Omron CX-Programmer project NewProject (CX-Programmer 9.51)

# PLC NewPLC1: CJ2M CPU11
I/O table (CPU CJ2M-CPU11): rack 0 slot 0 CJ1W-ID211; rack 0 slot 1 CJ1W-OD212; rack 0 slot 2 CJ1W-TC002; rack 0 slot 3 CJ1W-TC002; rack 0 slot 4 CJ1W-NC481; rack 0 slot 5 CJ1W-DA041; rack 0 slot 6 CJ1W-MAD42

## Global symbols (name address type ; comment)
AUX_AUTOMATICO W10.00 BOOL  ; Auxiliar maquina em Automático
AUX_LIMITE_NIPE W4.00 BOOL
AUX_MANUAL W10.01 BOOL  ; auxiliar maquina em trabalho manual
AUX_MANUAL_SERVO_NIP_LOCK W20.00 BOOL  ; Auxiliar para ligar manual do servo NIP
AUX_MANUAL_SERVO_NIP_UNLOCK W20.09 BOOL  ; Auxiliar UNLOCK servo NIP
AUX_MANUAL_SERVO_SEL_LOCK W20.02 BOOL  ; Auxiliar par ligar servo SEL
AUX_MANUAL_SERVO_SEL_UNLOCK W20.11 BOOL  ; Auxiliar para UNLOCK Servo SEL
AUX_MANUAL_SERVO_TRO_LOCK W20.01 BOOL  ; Auxiliar  para ligar servo TRO
AUX_MANUAL_SERVO_TRO_UNLOCK W20.10 BOOL  ; Auxiliar Unlock servo TRO
0.05 BOOL  ; Chave seletora Faca
0.13 BOOL  ; Botão Jog FACA avança
1.05 BOOL  ; INVERSOR DE PASSAGEM
1.12 BOOL  ; Saida habilita servo rebobinador inferior 2
1.13 BOOL  ; Saida Habililta servo rebobinador superior 2
2000.00 BOOL  ; Habilita Saída analógica 1
2000.01 BOOL  ; Habilita saída analógica 2
2030.00 BOOL  ; Habilita saída Rebobinador Superior 1
2030.01 BOOL  ; Habilita saída Rebobinador inferior 1
2030.02 BOOL  ; Habilita saída Rebobinador Superior 2
2030.03 BOOL  ; Habilita saída Rebobinador Inferior 2
2031 CHANNEL  ; Saída Analógica Rebobinador Superior
2032 CHANNEL  ; Saída Analógica Rebobinador  Inferior 1
2033 CHANNEL  ; Habilita saída Rebobinador Superior 2
2034 CHANNEL  ; Saída Analógica Rebobinador  Inferior 2
2040 CHANNEL  ; Setpoint da saída de aquecimento 5
A531.00 BOOL  ; ZERA CONTAGEM DO SENSOR
A531.01 BOOL  ; ZERA
D1012 CHANNEL  ; Posição do Corte
D1014 CHANNEL  ; Posição corte inferior
D104 CHANNEL  ; Valor para saida analógica reb sup 2
D106 CHANNEL  ; valor desejado de saida para rebobinador inferior 2
D124 CHANNEL  ; PRESET VALOR MIN DO TORQUE REB SUP 2
D126 CHANNEL  ; IHM preset valor min de torque para trabalho inferior2
D20 CHANNEL  ; CONT ETIQUETA
D200 CHANNEL  ; Controle Desbobinador Superior
D201 CHANNEL  ; Banda Proporcional Desbobinador superior
D202 CHANNEL  ; Constante Integral Desbobinador Superior
D203 CHANNEL  ; Constante Derivativo Desbobinador Superior
D204 CHANNEL  ; Tempo de Amostragem
D205 CHANNEL  ; Controle PID Desbobinador Sup
D206 CHANNEL  ; Controle PID Desbobinador Sup
D207 CHANNEL  ; Limite da variável manipulada
D209 CHANNEL  ; Controle PID automático e ganho
D210 CHANNEL  ; Histerese
D280 CHANNEL  ; Set Point Desbobinador Superior
D403 CHANNEL  ; IHM Constante selagem
D404 CHANNEL  ; IHM Constante Faca
D405 CHANNEL  ; FREIO DESBOBINADOR SUPERIOR
D406 CHANNEL  ; IHM Freio Desbobinador Inferior
D408 CHANNEL  ; IHM Tamanho do Pacote
D410 CHANNEL  ; IHM Velocidade Maquina M/min
D54 CHANNEL  ; IHM preset torque do Reb Sup 2, quando em automatico
D56 CHANNEL  ; IHM preset para torque Reb inf 2 quando a maquina estiver em trabalho
D700 CHANNEL  ; CONTANTE ACELERACAO
D701 CHANNEL  ; VELOCIDADE_ETQ
H0.00 BOOL  ; Seletora quantidade de facas
H45.00 BOOL  ; HABILITA ETIQUETA
T0002 BOOL  ; Tempo para acionamento do marcador
T0021 BOOL  ; Tempo para Reset
T0050 BOOL  ; ]
T0100 BOOL  ; Tempo Reset Ethercat
T0101 BOOL  ; Tempo para iniciar a verificação se chegou na origem
W1.00 BOOL  ; INDICA SERVOS LIGADOS
W1.02 BOOL  ; FLAG EM PRODUÇÃO
W1.03 BOOL  ; TRO REFERENCIADO
W200.00 BOOL  ; Aumento gradativo do torque
W20.03 BOOL  ; Auxiliar JOG NIP Horario
W20.04 BOOL  ; Auxiliar JOG NIP Anti-horario
W20.05 BOOL  ; Auxiliar JOG TRO Horario
W20.06 BOOL  ; Auxiliar JOG TRO Anti Horario
W20.07 BOOL  ; Auxiliar JOG SEL Horario
W20.08 BOOL  ; Auxiliar JOG SEL Anti horario
W2.03 BOOL  ; Auxiliar servos não estão em erro
W2.04 BOOL  ; Auxiliar Servos Lock
W2.05 BOOL  ; Auxiliar busca de origem
W33.00 BOOL  ; +
W33.01 BOOL  ; -
W3.00 BOOL  ; Flag Inicialização Completa
W50.07 BOOL  ; IHM botão liga servo Selagem
W50.08 BOOL  ; IHM botão liga servo TRO
W50.09 BOOL  ; IHM Botão Liga servo NIP Manual
W50.10 BOOL  ; IHM botão JOG SEL Horario
W50.11 BOOL  ; IHM botão JOG SEL Anti Horario
W50.12 BOOL  ; IHM botão JOG TRO Horario
W50.13 BOOL  ; IHM botão JOG TRO Anti Horario
W50.14 BOOL  ; IHM botão JOG NIP Horario
W50.15 BOOL  ; IHM botão JOG NIP Anti Horario
W60.04 BOOL  ; Botão Habilita servo Rebobinador superior 2
W60.05 BOOL  ; Botão Habilita servo Rebobinador inferior 2
W60.09 BOOL  ; IHM  Botão Reset
W60.10 BOOL  ; IHM PB busca da origem servo TRO
W60.11 BOOL  ; IHM Botão Liga/Desliga todos servos
W6.00 BOOL  ; PARA ROLDANA
W6.08 BOOL  ; SALVAR RECEITA
W6.09 BOOL  ; CARREGAR RECEITA
W6.12 BOOL  ; FLAG PERCA CORTE
W6.14 BOOL  ; MARCAR SENSOR
W7.00 BOOL  ; START AT1
W7.01 BOOL  ; START AT2
W7.02 BOOL  ; START AT3
W7.03 BOOL  ; START AT4
W7.04 BOOL  ; START AT5
W8.00 BOOL  ; MARCA SENSOR ETIQUETA
CH_SEL_LIGA_NIP 0.04 BOOL  ; Chave seletora para ligar acionamento do NIP
CH_SEL_MANUAL_AUTO 0.03 BOOL  ; Chave de seleção Manual ou Automático
CONTAGEM_ABS D670 CHANNEL  ; CONTAGEM_ABS
Calc_Sel Calc_Pacote
Calc_Tamanho_Pacote Calc_Pacote
Desbobinador_Sup Escala_SA
ETIQUETADOR CALC_ETIQUETA
IHM_Auto_Torque_Reb_Inf D52 REAL  ; IHM preset para torque rebobinador inferior quando a maquina estiver em trabalho
IHM_Auto_Torque_Reb_Sup D50 REAL  ; IHM preset torque do Rebobinador Superior, quando em automático
IHM_BT_FREIO_INF W60.01 BOOL
IHM_BT_FREIO_SUP W60.00 BOOL  ; Botão para acionamento no freio manual
IHM_BT_LOCK_REB_INF W60.03 BOOL  ; Botão Habilita servo Rebobinador inferior 1
IHM_BT_LOCK_REB_SUP W60.02 BOOL  ; Botão Habilita servo Rebobinador superior 1
IHM_Min_Reb_Inf D122 REAL  ; IHM preset valor minimo de torque para trabalho
IHM_Min_Reb_Sup D120 REAL  ; PRESET VALOR MINIMO DO TORQUE
IHM_PB_S_MARCADOR W50.03 BOOL  ; IHM Botão Acionamento manual do Etiquetador
IHM_PB_S_NIP W50.00 BOOL  ; IHM Botão acionamento manual do NIP
IHM_PB_S_NIP_SEL W50.02 BOOL  ; NIP Selagem
IHM_PB_S_SEL W50.01 BOOL  ; IHM Botão acionamento manual do tracionador Selagem
Inicializacao W0 CHANNEL  ; Controle inicialização
Inicializacao_passo_0 W0.00 BOOL
Inicializacao_passo_1 W0.01 BOOL
Inicializacao_passo_10 W0.10 BOOL
Inicializacao_passo_11 W0.11 BOOL
Inicializacao_passo_12 W0.12 BOOL
Inicializacao_passo_13 W0.13 BOOL
Inicializacao_passo_14 W0.14 BOOL
Inicializacao_passo_15 W0.15 BOOL
Inicializacao_passo_2 W0.02 BOOL
Inicializacao_passo_3 W0.03 BOOL
Inicializacao_passo_4 W0.04 BOOL
Inicializacao_passo_5 W0.05 BOOL
Inicializacao_passo_6 W0.06 BOOL
Inicializacao_passo_7 W0.07 BOOL
Inicializacao_passo_8 W0.08 BOOL
Inicializacao_passo_9 W0.09 BOOL
NCx8x_00_Axis1DirectOperation_AbsoluteMovementBit 3100.00 BOOL  ; AbsoluteMovementBit
NCx8x_00_Axis1DirectOperation_AccelerationTime 3108 DINT  ; AccelerationTime
NCx8x_00_Axis1DirectOperation_CommandPosition 3102 DINT  ; CommandPosition
NCx8x_00_Axis1DirectOperation_CommandSpeed 3104 DINT  ; CommandSpeed
NCx8x_00_Axis1DirectOperation_DecelerationTime 3110 DINT  ; DecelerationTime
NCx8x_00_Axis1DirectOperation_InterruptFeedingSpecificationBit 3100.05 BOOL  ; InterruptFeedingSpecificationBit
NCx8x_00_Axis1DirectOperation_InterruptInputMask_PresentPositionLatchEnableBit 3100.06 BOOL  ; InterruptInputMask_PresentPositionLatchEnableBit
NCx8x_00_Axis1DirectOperation_LatchCompletedFlagClearBit 3100.15 BOOL  ; LatchCompletedFlagClearBit
NCx8x_00_Axis1DirectOperation_OptionInput1 3106 UINT  ; OptionInput1
NCx8x_00_Axis1DirectOperation_OptionInput2 3107 UINT  ; OptionInput2
NCx8x_00_Axis1DirectOperation_OriginPositionLachCompletedFlagClearBit 3100.14 BOOL  ; OriginPositionLachCompletedFlagClearBit
NCx8x_00_Axis1DirectOperation_OriginPositionLachEnableBit 3100.11 BOOL  ; OriginPositionLachEnableBit
NCx8x_00_Axis1DirectOperation_PresentPositionPresetBit 3100.07 BOOL  ; PresentPositionPresetBit
NCx8x_00_Axis1DirectOperation_RelativeMovementBit 3100.01 BOOL  ; RelativeMovementBit
NCx8x_00_Axis1DirectOperation_RotationAxisDirection 3101 UINT  ; RotationAxisDirection
NCx8x_00_Axis1DirectOperation_SpeedControlBit 3100.02 BOOL  ; SpeedControlBit
NCx8x_00_Axis1ExpandedMonitor_ExpandedMonitor2 3500 DINT  ; ExpandedMonitor2
NCx8x_00_Axis1ExpandedMonitor_ExpandedMonitor3 3502 DINT  ; ExpandedMonitor3
NCx8x_00_Axis1ExpandedMonitor_ExpandedMonitor4 3504 DINT  ; ExpandedMonitor4
NCx8x_00_Axis1ExpandedMonitor_ExpandedMonitor5 3506 DINT  ; ExpandedMonitor5
NCx8x_00_Axis1ExpandedMonitor_ExpandedMonitor6 3508 DINT  ; ExpandedMonitor6
NCx8x_00_Axis1ManualOperation_DecelerationStopBit 3000.14 BOOL  ; DecelerationStopBit
NCx8x_00_Axis1ManualOperation_DeviationCounterResetBit 3000.02 BOOL  ; DeviationCounterResetBit
NCx8x_00_Axis1ManualOperation_DriveAlarmResetBit 3000.01 BOOL  ; DriveAlarmResetBit
NCx8x_00_Axis1ManualOperation_ForwardJogging_InchingBit 3000.07 BOOL  ; ForwardJogging_InchingBit
NCx8x_00_Axis1ManualOperation_ForwardTorqueLimitBit 3000.03 BOOL  ; ForwardTorqueLimitBit
NCx8x_00_Axis1ManualOperation_ImmediateStopBit 3000.13 BOOL  ; ImmediateStopBit
NCx8x_00_Axis1ManualOperation_Jogging_InchingSpeedSelectionBit 3000.06 BOOL  ; Jogging_InchingSpeedSelectionBit
NCx8x_00_Axis1ManualOperation_OriginReturnBit 3000.11 BOOL  ; OriginReturnBit
NCx8x_00_Axis1ManualOperation_OriginSearchBit 3000.10 BOOL  ; OriginSearchBit
NCx8x_00_Axis1ManualOperation_Override 3001 UINT  ; Override
NCx8x_00_Axis1ManualOperation_OverrideEnableBit 3000.05 BOOL  ; OverrideEnableBit
NCx8x_00_Axis1ManualOperation_ReverseJogging_InchingBit 3000.08 BOOL  ; ReverseJogging_InchingBit
NCx8x_00_Axis1ManualOperation_ReverseTorqueLimitBit 3000.04 BOOL  ; ReverseTorqueLimitBit
NCx8x_00_Axis1ManualOperation_ServoLockBit 3000.00 BOOL  ; ServoLockBit
NCx8x_00_Axis1ManualOperation_ServoUnlockBit 3000.15 BOOL  ; ServoUnlockBit
NCx8x_00_Axis1Status_AbsoluteMovementAcknowledgedFlag 3301.00 BOOL  ; AbsoluteMovementAcknowledgedFlag
NCx8x_00_Axis1Status_AbsoluteMovementFlag 3304.04 BOOL  ; AbsoluteMovementFlag
NCx8x_00_Axis1Status_AccelerationFlag 3303.03 BOOL  ; AccelerationFlag
NCx8x_00_Axis1Status_AlarmResetOutputFlag 3306.01 BOOL  ; AlarmResetOutputFlag
NCx8x_00_Axis1Status_AxisBusyFlag 3302.00 BOOL  ; AxisBusyFlag
NCx8x_00_Axis1Status_AxisErrorFlag 3305.12 BOOL  ; AxisErrorFlag
NCx8x_00_Axis1Status_AxisWarningFlag 3305.11 BOOL  ; AxisWarningFlag
NCx8x_00_Axis1Status_CommandPresentPosition 3308 DINT  ; CommandPresentPosition
NCx8x_00_Axis1Status_CommandPresentPositionOverflowFlag 3305.04 BOOL  ; CommandPresentPositionOverflowFlag
NCx8x_00_Axis1Status_CommandPresentPositionUnderflowFlag 3305.05 BOOL  ; CommandPresentPositionUnderflowFlag
NCx8x_00_Axis1Status_ConstantSpeedFlag 3303.04 BOOL  ; ConstantSpeedFlag
NCx8x_00_Axis1Status_DecelerationFlag 3303.05 BOOL  ; DecelerationFlag
NCx8x_00_Axis1Status_DecelerationStopAcknowledgedFlag 3300.14 BOOL  ; DecelerationStopAcknowledgedFlag
NCx8x_00_Axis1Status_DecelerationStopFlag 3303.08 BOOL  ; DecelerationStopFlag
NCx8x_00_Axis1Status_DeviationCounterResetAcknowledgedFlag 3300.02 BOOL  ; DeviationCounterResetAcknowledgedFlag
NCx8x_00_Axis1Status_DeviationCounterResetInvalidFlag 3302.09 BOOL  ; DeviationCounterResetInvalidFlag
NCx8x_00_Axis1Status_DeviationCounterResetOutputFlag 3306.02 BOOL  ; DeviationCounterResetOutputFlag
NCx8x_00_Axis1Status_DirectOperationEnabledFlag 3302.02 BOOL  ; DirectOperationEnabledFlag
NCx8x_00_Axis1Status_DriveAlarmInputFlag 3306.15 BOOL  ; DriveAlarmInputFlag
NCx8x_00_Axis1Status_DriveAlarmResetAcknowledgedFlag 3300.01 BOOL  ; DriveAlarmResetAcknowledgedFlag
NCx8x_00_Axis1Status_EmergencyStopInputFlag 3306.13 BOOL  ; EmergencyStopInputFlag
NCx8x_00_Axis1Status_ErrorCode 3307 UINT  ; ErrorCode
NCx8x_00_Axis1Status_ExecutionErrorFlag 3305.10 BOOL  ; ExecutionErrorFlag
NCx8x_00_Axis1Status_ExpandedMonitor 3310 DINT  ; ExpandedMonitor
NCx8x_00_Axis1Status_FeedbackPresentPositionOverflowFlag 3305.06 BOOL  ; FeedbackPresentPositionOverflowFlag
NCx8x_00_Axis1Status_FeedbackPresentPositionUnderflowFlag 3305.07 BOOL  ; FeedbackPresentPositionUnderflowFlag
NCx8x_00_Axis1Status_ForwardJogging_InchingAcknowledgedFlag 3300.07 BOOL  ; ForwardJogging_InchingAcknowledgedFlag
NCx8x_00_Axis1Status_ForwardLimitInputFlag 3306.08 BOOL  ; ForwardLimitInputFlag
NCx8x_00_Axis1Status_ForwardTorqueLimitAcknowledgedFlag 3300.03 BOOL  ; ForwardTorqueLimitAcknowledgedFlag
NCx8x_00_Axis1Status_ForwardTorqueLimitOutputFlag 3306.03 BOOL  ; ForwardTorqueLimitOutputFlag
NCx8x_00_Axis1Status_HighSpeedPTPStartAcknowledgedFlag 3302.07 BOOL  ; HighSpeedPTPStartAcknowledgedFlag
NCx8x_00_Axis1Status_ImmediateStopAcknowledgedFlag 3300.13 BOOL  ; ImmediateStopAcknowledgedFlag
NCx8x_00_Axis1Status_ImmediateStopFlag 3303.09 BOOL  ; ImmediateStopFlag
NCx8x_00_Axis1Status_InterruptFeedingSpecificationAcknowledgedFlag 3301.05 BOOL  ; InterruptFeedingSpecificationAcknowledgedFlag
NCx8x_00_Axis1Status_InterruptFeeding_InterruptInputWaitingFlag 3304.07 BOOL  ; InterruptFeeding_InterruptInputWaitingFlag
NCx8x_00_Axis1Status_InterruptFeeding_PositioningFlag 3304.08 BOOL  ; InterruptFeeding_PositioningFlag
NCx8x_00_Axis1Status_InterruptInputFlag 3306.12 BOOL  ; InterruptInputFlag
NCx8x_00_Axis1Status_InterruptInputMask_PresentPositionLatchEnableAcknowledgedFlag 3301.06 BOOL  ; InterruptInputMask_PresentPositionLatchEnableAcknowledgedFlag
NCx8x_00_Axis1Status_JoggingEnabledFlag 3302.01 BOOL  ; JoggingEnabledFlag
NCx8x_00_Axis1Status_Jogging_InchingFlag 3304.03 BOOL  ; Jogging_InchingFlag
NCx8x_00_Axis1Status_Jogging_InchingSpeedSelectionAcknowledgedFlag 3300.06 BOOL  ; Jogging_InchingSpeedSelectionAcknowledgedFlag
NCx8x_00_Axis1Status_LatchCompletedFlag 3305.02 BOOL  ; LatchCompletedFlag
NCx8x_00_Axis1Status_LatchCompletedFlagClearAcknowledgedFlag 3301.15 BOOL  ; LatchCompletedFlagClearAcknowledgedFlag
NCx8x_00_Axis1Status_MainCircuitStatusFlag 3306.05 BOOL  ; MainCircuitStatusFlag
NCx8x_00_Axis1Status_MemoryOperationFlag 3304.11 BOOL  ; MemoryOperationFlag
NCx8x_00_Axis1Status_OriginDefinedFlag 3305.00 BOOL  ; OriginDefinedFlag
NCx8x_00_Axis1Status_OriginInputFlag 3306.11 BOOL  ; OriginInputFlag
NCx8x_00_Axis1Status_OriginPositionLatchCompletedFlag 3305.03 BOOL  ; OriginPositionLatchCompletedFlag
NCx8x_00_Axis1Status_OriginPositionLatchCompletedFlagClearAcknowledgedFlag 3301.14 BOOL  ; OriginPositionLatchCompletedFlagClearAcknowledgedFlag
NCx8x_00_Axis1Status_OriginPositionLatchEnableAcknowledgedFlag 3301.11 BOOL  ; OriginPositionLatchEnableAcknowledgedFlag
NCx8x_00_Axis1Status_OriginProximityInputFlag 3306.10 BOOL  ; OriginProximityInputFlag
NCx8x_00_Axis1Status_OriginReturnAcknowledgedFlag 3300.11 BOOL  ; OriginReturnAcknowledgedFlag
NCx8x_00_Axis1Status_OriginReturnFlag 3304.01 BOOL  ; OriginReturnFlag
NCx8x_00_Axis1Status_OriginSearchAcknowledgedFlag 3300.10 BOOL  ; OriginSearchAcknowledgedFlag
NCx8x_00_Axis1Status_OriginSearchFlag 3304.00 BOOL  ; OriginSearchFlag
NCx8x_00_Axis1Status_OverrideEnableAcknowledgedFlag 3300.05 BOOL  ; OverrideEnableAcknowledgedFlag
NCx8x_00_Axis1Status_PassFlag 3303.06 BOOL  ; PassFlag
NCx8x_00_Axis1Status_PositioningCompletedInputFlag 3306.14 BOOL  ; PositioningCompletedInputFlag
NCx8x_00_Axis1Status_PositioningCompletedWaitingFlag 3303.07 BOOL  ; PositioningCompletedWaitingFlag
NCx8x_00_Axis1Status_PositioningOperationCompletedFlag 3302.13 BOOL  ; PositioningOperationCompletedFlag
NCx8x_00_Axis1Status_PresentPositionPresetAcknowledgedFlag 3301.07 BOOL  ; PresentPositionPresetAcknowledgedFlag
NCx8x_00_Axis1Status_RelativeMovementAcknowledgedFlag 3301.01 BOOL  ; RelativeMovementAcknowledgedFlag
NCx8x_00_Axis1Status_RelativeMovementFlag 3304.05 BOOL  ; RelativeMovementFlag
NCx8x_00_Axis1Status_ReverseJogging_InchingAcknowledgedFlag 3300.08 BOOL  ; ReverseJogging_InchingAcknowledgedFlag
NCx8x_00_Axis1Status_ReverseLimitInputFlag 3306.09 BOOL  ; ReverseLimitInputFlag
NCx8x_00_Axis1Status_ReverseTorqueLimitAcknowledgedFlag 3300.04 BOOL  ; ReverseTorqueLimitAcknowledgedFlag
NCx8x_00_Axis1Status_ReverseTorqueLimitOutputFlag 3306.04 BOOL  ; ReverseTorqueLimitOutputFlag
NCx8x_00_Axis1Status_SensorErrorFlag 3305.08 BOOL  ; SensorErrorFlag
NCx8x_00_Axis1Status_ServoDriveWarningFlag 3306.06 BOOL  ; ServoDriveWarningFlag
NCx8x_00_Axis1Status_ServoErrorFlag 3305.09 BOOL  ; ServoErrorFlag
NCx8x_00_Axis1Status_ServoLockAcknowledgedFlag 3300.00 BOOL  ; ServoLockAcknowledgedFlag
NCx8x_00_Axis1Status_ServoLockedFlag 3303.01 BOOL  ; ServoLockedFlag
NCx8x_00_Axis1Status_ServoONFlag 3306.00 BOOL  ; ServoONFlag
NCx8x_00_Axis1Status_ServoReadyFlag 3306.07 BOOL  ; ServoReadyFlag
NCx8x_00_Axis1Status_ServoUnlockAcknowledgedFlag 3300.15 BOOL  ; ServoUnlockAcknowledgedFlag
NCx8x_00_Axis1Status_ServoUnlockedFlag 3303.00 BOOL  ; ServoUnlockedFlag
NCx8x_00_Axis1Status_SpeedControlAcknowledgedFlag 3301.02 BOOL  ; SpeedControlAcknowledgedFlag
NCx8x_00_Axis1Status_SpeedControlFlag 3304.06 BOOL  ; SpeedControlFlag
NCx8x_00_Axis1Status_StartInvalidFlag 3302.08 BOOL  ; StartInvalidFlag
NCx8x_00_Axis1Status_StopExecutedFlag 3302.12 BOOL  ; StopExecutedFlag
NCx8x_00_Axis1Status_StopInputFlag 3302.04 BOOL  ; StopInputFlag
NCx8x_00_Axis1Status_StoppedatOriginFlag 3305.01 BOOL  ; StoppedatOriginFlag
NCx8x_00_Axis1Status_Zone0Flag 3305.13 BOOL  ; Zone0Flag
NCx8x_00_Axis1Status_Zone1Flag 3305.14 BOOL  ; Zone1Flag
NCx8x_00_Axis1Status_Zone2Flag 3305.15 BOOL  ; Zone2Flag
NCx8x_00_Axis2DirectOperation_AbsoluteMovementBit 3112.00 BOOL  ; AbsoluteMovementBit
NCx8x_00_Axis2DirectOperation_AccelerationTime 3120 DINT  ; AccelerationTime
NCx8x_00_Axis2DirectOperation_CommandPosition 3114 DINT  ; CommandPosition
NCx8x_00_Axis2DirectOperation_CommandSpeed 3116 DINT  ; CommandSpeed
NCx8x_00_Axis2DirectOperation_DecelerationTime 3122 DINT  ; DecelerationTime
NCx8x_00_Axis2DirectOperation_InterruptFeedingSpecificationBit 3112.05 BOOL  ; InterruptFeedingSpecificationBit
NCx8x_00_Axis2DirectOperation_InterruptInputMask_PresentPositionLatchEnableBit 3112.06 BOOL  ; InterruptInputMask_PresentPositionLatchEnableBit
NCx8x_00_Axis2DirectOperation_LatchCompletedFlagClearBit 3112.15 BOOL  ; LatchCompletedFlagClearBit
NCx8x_00_Axis2DirectOperation_OptionInput1 3118 UINT  ; OptionInput1
NCx8x_00_Axis2DirectOperation_OptionInput2 3119 UINT  ; OptionInput2
NCx8x_00_Axis2DirectOperation_OriginPositionLachCompletedFlagClearBit 3112.14 BOOL  ; OriginPositionLachCompletedFlagClearBit
NCx8x_00_Axis2DirectOperation_OriginPositionLachEnableBit 3112.11 BOOL  ; OriginPositionLachEnableBit
NCx8x_00_Axis2DirectOperation_PresentPositionPresetBit 3112.07 BOOL  ; PresentPositionPresetBit
NCx8x_00_Axis2DirectOperation_RelativeMovementBit 3112.01 BOOL  ; RelativeMovementBit
NCx8x_00_Axis2DirectOperation_RotationAxisDirection 3113 UINT  ; RotationAxisDirection
NCx8x_00_Axis2DirectOperation_SpeedControlBit 3112.02 BOOL  ; SpeedControlBit
NCx8x_00_Axis2ExpandedMonitor_ExpandedMonitor2 3516 DINT  ; ExpandedMonitor2
NCx8x_00_Axis2ExpandedMonitor_ExpandedMonitor3 3518 DINT  ; ExpandedMonitor3
NCx8x_00_Axis2ExpandedMonitor_ExpandedMonitor4 3520 DINT  ; ExpandedMonitor4
NCx8x_00_Axis2ExpandedMonitor_ExpandedMonitor5 3522 DINT  ; ExpandedMonitor5
NCx8x_00_Axis2ExpandedMonitor_ExpandedMonitor6 3524 DINT  ; ExpandedMonitor6
NCx8x_00_Axis2ManualOperation_DecelerationStopBit 3002.14 BOOL  ; DecelerationStopBit
NCx8x_00_Axis2ManualOperation_DeviationCounterResetBit 3002.02 BOOL  ; DeviationCounterResetBit
NCx8x_00_Axis2ManualOperation_DriveAlarmResetBit 3002.01 BOOL  ; DriveAlarmResetBit
NCx8x_00_Axis2ManualOperation_ForwardJogging_InchingBit 3002.07 BOOL  ; ForwardJogging_InchingBit
NCx8x_00_Axis2ManualOperation_ForwardTorqueLimitBit 3002.03 BOOL  ; ForwardTorqueLimitBit
NCx8x_00_Axis2ManualOperation_ImmediateStopBit 3002.13 BOOL  ; ImmediateStopBit
NCx8x_00_Axis2ManualOperation_Jogging_InchingSpeedSelectionBit 3002.06 BOOL  ; Jogging_InchingSpeedSelectionBit
NCx8x_00_Axis2ManualOperation_OriginReturnBit 3002.11 BOOL  ; OriginReturnBit
NCx8x_00_Axis2ManualOperation_OriginSearchBit 3002.10 BOOL  ; OriginSearchBit
NCx8x_00_Axis2ManualOperation_Override 3003 UINT  ; Override
NCx8x_00_Axis2ManualOperation_OverrideEnableBit 3002.05 BOOL  ; OverrideEnableBit
NCx8x_00_Axis2ManualOperation_ReverseJogging_InchingBit 3002.08 BOOL  ; ReverseJogging_InchingBit
NCx8x_00_Axis2ManualOperation_ReverseTorqueLimitBit 3002.04 BOOL  ; ReverseTorqueLimitBit
NCx8x_00_Axis2ManualOperation_ServoLockBit 3002.00 BOOL  ; ServoLockBit
NCx8x_00_Axis2ManualOperation_ServoUnlockBit 3002.15 BOOL  ; ServoUnlockBit
NCx8x_00_Axis2Status_AbsoluteMovementAcknowledgedFlag 3314.00 BOOL  ; AbsoluteMovementAcknowledgedFlag
NCx8x_00_Axis2Status_AbsoluteMovementFlag 3317.04 BOOL  ; AbsoluteMovementFlag
NCx8x_00_Axis2Status_AccelerationFlag 3316.03 BOOL  ; AccelerationFlag
NCx8x_00_Axis2Status_AlarmResetOutputFlag 3319.01 BOOL  ; AlarmResetOutputFlag
NCx8x_00_Axis2Status_AxisBusyFlag 3315.00 BOOL  ; AxisBusyFlag
NCx8x_00_Axis2Status_AxisErrorFlag 3318.12 BOOL  ; AxisErrorFlag
NCx8x_00_Axis2Status_AxisWarningFlag 3318.11 BOOL  ; AxisWarningFlag
NCx8x_00_Axis2Status_CommandPresentPosition 3321 DINT  ; CommandPresentPosition
NCx8x_00_Axis2Status_CommandPresentPositionOverflowFlag 3318.04 BOOL  ; CommandPresentPositionOverflowFlag
NCx8x_00_Axis2Status_CommandPresentPositionUnderflowFlag 3318.05 BOOL  ; CommandPresentPositionUnderflowFlag
NCx8x_00_Axis2Status_ConstantSpeedFlag 3316.04 BOOL  ; ConstantSpeedFlag
NCx8x_00_Axis2Status_DecelerationFlag 3316.05 BOOL  ; DecelerationFlag
NCx8x_00_Axis2Status_DecelerationStopAcknowledgedFlag 3313.14 BOOL  ; DecelerationStopAcknowledgedFlag
NCx8x_00_Axis2Status_DecelerationStopFlag 3316.08 BOOL  ; DecelerationStopFlag
NCx8x_00_Axis2Status_DeviationCounterResetAcknowledgedFlag 3313.02 BOOL  ; DeviationCounterResetAcknowledgedFlag
NCx8x_00_Axis2Status_DeviationCounterResetInvalidFlag 3315.09 BOOL  ; DeviationCounterResetInvalidFlag
NCx8x_00_Axis2Status_DeviationCounterResetOutputFlag 3319.02 BOOL  ; DeviationCounterResetOutputFlag
NCx8x_00_Axis2Status_DirectOperationEnabledFlag 3315.02 BOOL  ; DirectOperationEnabledFlag
NCx8x_00_Axis2Status_DriveAlarmInputFlag 3319.15 BOOL  ; DriveAlarmInputFlag
NCx8x_00_Axis2Status_DriveAlarmResetAcknowledgedFlag 3313.01 BOOL  ; DriveAlarmResetAcknowledgedFlag
NCx8x_00_Axis2Status_EmergencyStopInputFlag 3319.13 BOOL  ; EmergencyStopInputFlag
NCx8x_00_Axis2Status_ErrorCode 3320 UINT  ; ErrorCode
NCx8x_00_Axis2Status_ExecutionErrorFlag 3318.10 BOOL  ; ExecutionErrorFlag
NCx8x_00_Axis2Status_ExpandedMonitor 3323 DINT  ; ExpandedMonitor
NCx8x_00_Axis2Status_FeedbackPresentPositionOverflowFlag 3318.06 BOOL  ; FeedbackPresentPositionOverflowFlag
NCx8x_00_Axis2Status_FeedbackPresentPositionUnderflowFlag 3318.07 BOOL  ; FeedbackPresentPositionUnderflowFlag
NCx8x_00_Axis2Status_ForwardJogging_InchingAcknowledgedFlag 3313.07 BOOL  ; ForwardJogging_InchingAcknowledgedFlag
NCx8x_00_Axis2Status_ForwardLimitInputFlag 3319.08 BOOL  ; ForwardLimitInputFlag
NCx8x_00_Axis2Status_ForwardTorqueLimitAcknowledgedFlag 3313.03 BOOL  ; ForwardTorqueLimitAcknowledgedFlag
NCx8x_00_Axis2Status_ForwardTorqueLimitOutputFlag 3319.03 BOOL  ; ForwardTorqueLimitOutputFlag
NCx8x_00_Axis2Status_HighSpeedPTPStartAcknowledgedFlag 3315.07 BOOL  ; HighSpeedPTPStartAcknowledgedFlag
NCx8x_00_Axis2Status_ImmediateStopAcknowledgedFlag 3313.13 BOOL  ; ImmediateStopAcknowledgedFlag
NCx8x_00_Axis2Status_ImmediateStopFlag 3316.09 BOOL  ; ImmediateStopFlag
NCx8x_00_Axis2Status_InterruptFeedingSpecificationAcknowledgedFlag 3314.05 BOOL  ; InterruptFeedingSpecificationAcknowledgedFlag
NCx8x_00_Axis2Status_InterruptFeeding_InterruptInputWaitingFlag 3317.07 BOOL  ; InterruptFeeding_InterruptInputWaitingFlag
NCx8x_00_Axis2Status_InterruptFeeding_PositioningFlag 3317.08 BOOL  ; InterruptFeeding_PositioningFlag
NCx8x_00_Axis2Status_InterruptInputFlag 3319.12 BOOL  ; InterruptInputFlag
NCx8x_00_Axis2Status_InterruptInputMask_PresentPositionLatchEnableAcknowledgedFlag 3314.06 BOOL  ; InterruptInputMask_PresentPositionLatchEnableAcknowledgedFlag
NCx8x_00_Axis2Status_JoggingEnabledFlag 3315.01 BOOL  ; JoggingEnabledFlag
NCx8x_00_Axis2Status_Jogging_InchingFlag 3317.03 BOOL  ; Jogging_InchingFlag
NCx8x_00_Axis2Status_Jogging_InchingSpeedSelectionAcknowledgedFlag 3313.06 BOOL  ; Jogging_InchingSpeedSelectionAcknowledgedFlag
NCx8x_00_Axis2Status_LatchCompletedFlag 3318.02 BOOL  ; LatchCompletedFlag
NCx8x_00_Axis2Status_LatchCompletedFlagClearAcknowledgedFlag 3314.15 BOOL  ; LatchCompletedFlagClearAcknowledgedFlag
NCx8x_00_Axis2Status_MainCircuitStatusFlag 3319.05 BOOL  ; MainCircuitStatusFlag
NCx8x_00_Axis2Status_MemoryOperationFlag 3317.11 BOOL  ; MemoryOperationFlag
NCx8x_00_Axis2Status_OriginDefinedFlag 3318.00 BOOL  ; OriginDefinedFlag
NCx8x_00_Axis2Status_OriginInputFlag 3319.11 BOOL  ; OriginInputFlag
NCx8x_00_Axis2Status_OriginPositionLatchCompletedFlag 3318.03 BOOL  ; OriginPositionLatchCompletedFlag
NCx8x_00_Axis2Status_OriginPositionLatchCompletedFlagClearAcknowledgedFlag 3314.14 BOOL  ; OriginPositionLatchCompletedFlagClearAcknowledgedFlag
NCx8x_00_Axis2Status_OriginPositionLatchEnableAcknowledgedFlag 3314.11 BOOL  ; OriginPositionLatchEnableAcknowledgedFlag
NCx8x_00_Axis2Status_OriginProximityInputFlag 3319.10 BOOL  ; OriginProximityInputFlag
NCx8x_00_Axis2Status_OriginReturnAcknowledgedFlag 3313.11 BOOL  ; OriginReturnAcknowledgedFlag
NCx8x_00_Axis2Status_OriginReturnFlag 3317.01 BOOL  ; OriginReturnFlag
NCx8x_00_Axis2Status_OriginSearchAcknowledgedFlag 3313.10 BOOL  ; OriginSearchAcknowledgedFlag
NCx8x_00_Axis2Status_OriginSearchFlag 3317.00 BOOL  ; OriginSearchFlag
NCx8x_00_Axis2Status_OverrideEnableAcknowledgedFlag 3313.05 BOOL  ; OverrideEnableAcknowledgedFlag
NCx8x_00_Axis2Status_PassFlag 3316.06 BOOL  ; PassFlag
NCx8x_00_Axis2Status_PositioningCompletedInputFlag 3319.14 BOOL  ; PositioningCompletedInputFlag
NCx8x_00_Axis2Status_PositioningCompletedWaitingFlag 3316.07 BOOL  ; PositioningCompletedWaitingFlag
NCx8x_00_Axis2Status_PositioningOperationCompletedFlag 3315.13 BOOL  ; PositioningOperationCompletedFlag
NCx8x_00_Axis2Status_PresentPositionPresetAcknowledgedFlag 3314.07 BOOL  ; PresentPositionPresetAcknowledgedFlag
NCx8x_00_Axis2Status_RelativeMovementAcknowledgedFlag 3314.01 BOOL  ; RelativeMovementAcknowledgedFlag
NCx8x_00_Axis2Status_RelativeMovementFlag 3317.05 BOOL  ; RelativeMovementFlag
NCx8x_00_Axis2Status_ReverseJogging_InchingAcknowledgedFlag 3313.08 BOOL  ; ReverseJogging_InchingAcknowledgedFlag
NCx8x_00_Axis2Status_ReverseLimitInputFlag 3319.09 BOOL  ; ReverseLimitInputFlag
NCx8x_00_Axis2Status_ReverseTorqueLimitAcknowledgedFlag 3313.04 BOOL  ; ReverseTorqueLimitAcknowledgedFlag
NCx8x_00_Axis2Status_ReverseTorqueLimitOutputFlag 3319.04 BOOL  ; ReverseTorqueLimitOutputFlag
NCx8x_00_Axis2Status_SensorErrorFlag 3318.08 BOOL  ; SensorErrorFlag
NCx8x_00_Axis2Status_ServoDriveWarningFlag 3319.06 BOOL  ; ServoDriveWarningFlag
NCx8x_00_Axis2Status_ServoErrorFlag 3318.09 BOOL  ; ServoErrorFlag
NCx8x_00_Axis2Status_ServoLockAcknowledgedFlag 3313.00 BOOL  ; ServoLockAcknowledgedFlag
NCx8x_00_Axis2Status_ServoLockedFlag 3316.01 BOOL  ; ServoLockedFlag
NCx8x_00_Axis2Status_ServoONFlag 3319.00 BOOL  ; ServoONFlag
NCx8x_00_Axis2Status_ServoReadyFlag 3319.07 BOOL  ; ServoReadyFlag
NCx8x_00_Axis2Status_ServoUnlockAcknowledgedFlag 3313.15 BOOL  ; ServoUnlockAcknowledgedFlag
NCx8x_00_Axis2Status_ServoUnlockedFlag 3316.00 BOOL  ; ServoUnlockedFlag
NCx8x_00_Axis2Status_SpeedControlAcknowledgedFlag 3314.02 BOOL  ; SpeedControlAcknowledgedFlag
NCx8x_00_Axis2Status_SpeedControlFlag 3317.06 BOOL  ; SpeedControlFlag
NCx8x_00_Axis2Status_StartInvalidFlag 3315.08 BOOL  ; StartInvalidFlag
NCx8x_00_Axis2Status_StopExecutedFlag 3315.12 BOOL  ; StopExecutedFlag
NCx8x_00_Axis2Status_StopInputFlag 3315.04 BOOL  ; StopInputFlag
NCx8x_00_Axis2Status_StoppedatOriginFlag 3318.01 BOOL  ; StoppedatOriginFlag
NCx8x_00_Axis2Status_Zone0Flag 3318.13 BOOL  ; Zone0Flag
NCx8x_00_Axis2Status_Zone1Flag 3318.14 BOOL  ; Zone1Flag
NCx8x_00_Axis2Status_Zone2Flag 3318.15 BOOL  ; Zone2Flag
NCx8x_00_Axis3DirectOperation_AbsoluteMovementBit 3124.00 BOOL  ; AbsoluteMovementBit
NCx8x_00_Axis3DirectOperation_AccelerationTime 3132 DINT  ; AccelerationTime
NCx8x_00_Axis3DirectOperation_CommandPosition 3126 DINT  ; CommandPosition
NCx8x_00_Axis3DirectOperation_CommandSpeed 3128 DINT  ; CommandSpeed
NCx8x_00_Axis3DirectOperation_DecelerationTime 3134 DINT  ; DecelerationTime
NCx8x_00_Axis3DirectOperation_InterruptFeedingSpecificationBit 3124.05 BOOL  ; InterruptFeedingSpecificationBit
NCx8x_00_Axis3DirectOperation_InterruptInputMask_PresentPositionLatchEnableBit 3124.06 BOOL  ; InterruptInputMask_PresentPositionLatchEnableBit
NCx8x_00_Axis3DirectOperation_LatchCompletedFlagClearBit 3124.15 BOOL  ; LatchCompletedFlagClearBit
NCx8x_00_Axis3DirectOperation_OptionInput1 3130 UINT  ; OptionInput1
NCx8x_00_Axis3DirectOperation_OptionInput2 3131 UINT  ; OptionInput2
NCx8x_00_Axis3DirectOperation_OriginPositionLachCompletedFlagClearBit 3124.14 BOOL  ; OriginPositionLachCompletedFlagClearBit
NCx8x_00_Axis3DirectOperation_OriginPositionLachEnableBit 3124.11 BOOL  ; OriginPositionLachEnableBit
NCx8x_00_Axis3DirectOperation_PresentPositionPresetBit 3124.07 BOOL  ; PresentPositionPresetBit
NCx8x_00_Axis3DirectOperation_RelativeMovementBit 3124.01 BOOL  ; RelativeMovementBit
NCx8x_00_Axis3DirectOperation_RotationAxisDirection 3125 UINT  ; RotationAxisDirection
NCx8x_00_Axis3DirectOperation_SpeedControlBit 3124.02 BOOL  ; SpeedControlBit
NCx8x_00_Axis3ExpandedMonitor_ExpandedMonitor2 3532 DINT  ; ExpandedMonitor2
NCx8x_00_Axis3ExpandedMonitor_ExpandedMonitor3 3534 DINT  ; ExpandedMonitor3
NCx8x_00_Axis3ExpandedMonitor_ExpandedMonitor4 3536 DINT  ; ExpandedMonitor4
NCx8x_00_Axis3ExpandedMonitor_ExpandedMonitor5 3538 DINT  ; ExpandedMonitor5
NCx8x_00_Axis3ExpandedMonitor_ExpandedMonitor6 3540 DINT  ; ExpandedMonitor6
NCx8x_00_Axis3ManualOperation_DecelerationStopBit 3004.14 BOOL  ; DecelerationStopBit
NCx8x_00_Axis3ManualOperation_DeviationCounterResetBit 3004.02 BOOL  ; DeviationCounterResetBit
NCx8x_00_Axis3ManualOperation_DriveAlarmResetBit 3004.01 BOOL  ; DriveAlarmResetBit
NCx8x_00_Axis3ManualOperation_ForwardJogging_InchingBit 3004.07 BOOL  ; ForwardJogging_InchingBit
NCx8x_00_Axis3ManualOperation_ForwardTorqueLimitBit 3004.03 BOOL  ; ForwardTorqueLimitBit
NCx8x_00_Axis3ManualOperation_ImmediateStopBit 3004.13 BOOL  ; ImmediateStopBit
NCx8x_00_Axis3ManualOperation_Jogging_InchingSpeedSelectionBit 3004.06 BOOL  ; Jogging_InchingSpeedSelectionBit
NCx8x_00_Axis3ManualOperation_OriginReturnBit 3004.11 BOOL  ; OriginReturnBit
NCx8x_00_Axis3ManualOperation_OriginSearchBit 3004.10 BOOL  ; OriginSearchBit
NCx8x_00_Axis3ManualOperation_Override 3005 UINT  ; Override
NCx8x_00_Axis3ManualOperation_OverrideEnableBit 3004.05 BOOL  ; OverrideEnableBit
NCx8x_00_Axis3ManualOperation_ReverseJogging_InchingBit 3004.08 BOOL  ; ReverseJogging_InchingBit
NCx8x_00_Axis3ManualOperation_ReverseTorqueLimitBit 3004.04 BOOL  ; ReverseTorqueLimitBit
NCx8x_00_Axis3ManualOperation_ServoLockBit 3004.00 BOOL  ; ServoLockBit
NCx8x_00_Axis3ManualOperation_ServoUnlockBit 3004.15 BOOL  ; ServoUnlockBit
NCx8x_00_Axis3Status_AbsoluteMovementAcknowledgedFlag 3327.00 BOOL  ; AbsoluteMovementAcknowledgedFlag
NCx8x_00_Axis3Status_AbsoluteMovementFlag 3330.04 BOOL  ; AbsoluteMovementFlag
NCx8x_00_Axis3Status_AccelerationFlag 3329.03 BOOL  ; AccelerationFlag
NCx8x_00_Axis3Status_AlarmResetOutputFlag 3332.01 BOOL  ; AlarmResetOutputFlag
NCx8x_00_Axis3Status_AxisBusyFlag 3328.00 BOOL  ; AxisBusyFlag
NCx8x_00_Axis3Status_AxisErrorFlag 3331.12 BOOL  ; AxisErrorFlag
NCx8x_00_Axis3Status_AxisWarningFlag 3331.11 BOOL  ; AxisWarningFlag
NCx8x_00_Axis3Status_CommandPresentPosition 3334 DINT  ; CommandPresentPosition
NCx8x_00_Axis3Status_CommandPresentPositionOverflowFlag 3331.04 BOOL  ; CommandPresentPositionOverflowFlag
NCx8x_00_Axis3Status_CommandPresentPositionUnderflowFlag 3331.05 BOOL  ; CommandPresentPositionUnderflowFlag
NCx8x_00_Axis3Status_ConstantSpeedFlag 3329.04 BOOL  ; ConstantSpeedFlag
NCx8x_00_Axis3Status_DecelerationFlag 3329.05 BOOL  ; DecelerationFlag
NCx8x_00_Axis3Status_DecelerationStopAcknowledgedFlag 3326.14 BOOL  ; DecelerationStopAcknowledgedFlag
NCx8x_00_Axis3Status_DecelerationStopFlag 3329.08 BOOL  ; DecelerationStopFlag
NCx8x_00_Axis3Status_DeviationCounterResetAcknowledgedFlag 3326.02 BOOL  ; DeviationCounterResetAcknowledgedFlag
NCx8x_00_Axis3Status_DeviationCounterResetInvalidFlag 3328.09 BOOL  ; DeviationCounterResetInvalidFlag
NCx8x_00_Axis3Status_DeviationCounterResetOutputFlag 3332.02 BOOL  ; DeviationCounterResetOutputFlag
NCx8x_00_Axis3Status_DirectOperationEnabledFlag 3328.02 BOOL  ; DirectOperationEnabledFlag
NCx8x_00_Axis3Status_DriveAlarmInputFlag 3332.15 BOOL  ; DriveAlarmInputFlag
NCx8x_00_Axis3Status_DriveAlarmResetAcknowledgedFlag 3326.01 BOOL  ; DriveAlarmResetAcknowledgedFlag
NCx8x_00_Axis3Status_EmergencyStopInputFlag 3332.13 BOOL  ; EmergencyStopInputFlag
NCx8x_00_Axis3Status_ErrorCode 3333 UINT  ; ErrorCode
NCx8x_00_Axis3Status_ExecutionErrorFlag 3331.10 BOOL  ; ExecutionErrorFlag
NCx8x_00_Axis3Status_ExpandedMonitor 3336 DINT  ; ExpandedMonitor
NCx8x_00_Axis3Status_FeedbackPresentPositionOverflowFlag 3331.06 BOOL  ; FeedbackPresentPositionOverflowFlag
NCx8x_00_Axis3Status_FeedbackPresentPositionUnderflowFlag 3331.07 BOOL  ; FeedbackPresentPositionUnderflowFlag
NCx8x_00_Axis3Status_ForwardJogging_InchingAcknowledgedFlag 3326.07 BOOL  ; ForwardJogging_InchingAcknowledgedFlag
NCx8x_00_Axis3Status_ForwardLimitInputFlag 3332.08 BOOL  ; ForwardLimitInputFlag
NCx8x_00_Axis3Status_ForwardTorqueLimitAcknowledgedFlag 3326.03 BOOL  ; ForwardTorqueLimitAcknowledgedFlag
NCx8x_00_Axis3Status_ForwardTorqueLimitOutputFlag 3332.03 BOOL  ; ForwardTorqueLimitOutputFlag
NCx8x_00_Axis3Status_HighSpeedPTPStartAcknowledgedFlag 3328.07 BOOL  ; HighSpeedPTPStartAcknowledgedFlag
NCx8x_00_Axis3Status_ImmediateStopAcknowledgedFlag 3326.13 BOOL  ; ImmediateStopAcknowledgedFlag
NCx8x_00_Axis3Status_ImmediateStopFlag 3329.09 BOOL  ; ImmediateStopFlag
NCx8x_00_Axis3Status_InterruptFeedingSpecificationAcknowledgedFlag 3327.05 BOOL  ; InterruptFeedingSpecificationAcknowledgedFlag
NCx8x_00_Axis3Status_InterruptFeeding_InterruptInputWaitingFlag 3330.07 BOOL  ; InterruptFeeding_InterruptInputWaitingFlag
NCx8x_00_Axis3Status_InterruptFeeding_PositioningFlag 3330.08 BOOL  ; InterruptFeeding_PositioningFlag
NCx8x_00_Axis3Status_InterruptInputFlag 3332.12 BOOL  ; InterruptInputFlag
NCx8x_00_Axis3Status_InterruptInputMask_PresentPositionLatchEnableAcknowledgedFlag 3327.06 BOOL  ; InterruptInputMask_PresentPositionLatchEnableAcknowledgedFlag
NCx8x_00_Axis3Status_JoggingEnabledFlag 3328.01 BOOL  ; JoggingEnabledFlag
NCx8x_00_Axis3Status_Jogging_InchingFlag 3330.03 BOOL  ; Jogging_InchingFlag
NCx8x_00_Axis3Status_Jogging_InchingSpeedSelectionAcknowledgedFlag 3326.06 BOOL  ; Jogging_InchingSpeedSelectionAcknowledgedFlag
NCx8x_00_Axis3Status_LatchCompletedFlag 3331.02 BOOL  ; LatchCompletedFlag
NCx8x_00_Axis3Status_LatchCompletedFlagClearAcknowledgedFlag 3327.15 BOOL  ; LatchCompletedFlagClearAcknowledgedFlag
NCx8x_00_Axis3Status_MainCircuitStatusFlag 3332.05 BOOL  ; MainCircuitStatusFlag
NCx8x_00_Axis3Status_MemoryOperationFlag 3330.11 BOOL  ; MemoryOperationFlag
NCx8x_00_Axis3Status_OriginDefinedFlag 3331.00 BOOL  ; OriginDefinedFlag
NCx8x_00_Axis3Status_OriginInputFlag 3332.11 BOOL  ; OriginInputFlag
NCx8x_00_Axis3Status_OriginPositionLatchCompletedFlag 3331.03 BOOL  ; OriginPositionLatchCompletedFlag
NCx8x_00_Axis3Status_OriginPositionLatchCompletedFlagClearAcknowledgedFlag 3327.14 BOOL  ; OriginPositionLatchCompletedFlagClearAcknowledgedFlag
NCx8x_00_Axis3Status_OriginPositionLatchEnableAcknowledgedFlag 3327.11 BOOL  ; OriginPositionLatchEnableAcknowledgedFlag
NCx8x_00_Axis3Status_OriginProximityInputFlag 3332.10 BOOL  ; OriginProximityInputFlag
NCx8x_00_Axis3Status_OriginReturnAcknowledgedFlag 3326.11 BOOL  ; OriginReturnAcknowledgedFlag
NCx8x_00_Axis3Status_OriginReturnFlag 3330.01 BOOL  ; OriginReturnFlag
NCx8x_00_Axis3Status_OriginSearchAcknowledgedFlag 3326.10 BOOL  ; OriginSearchAcknowledgedFlag
NCx8x_00_Axis3Status_OriginSearchFlag 3330.00 BOOL  ; OriginSearchFlag
NCx8x_00_Axis3Status_OverrideEnableAcknowledgedFlag 3326.05 BOOL  ; OverrideEnableAcknowledgedFlag
NCx8x_00_Axis3Status_PassFlag 3329.06 BOOL  ; PassFlag
NCx8x_00_Axis3Status_PositioningCompletedInputFlag 3332.14 BOOL  ; PositioningCompletedInputFlag
NCx8x_00_Axis3Status_PositioningCompletedWaitingFlag 3329.07 BOOL  ; PositioningCompletedWaitingFlag
NCx8x_00_Axis3Status_PositioningOperationCompletedFlag 3328.13 BOOL  ; PositioningOperationCompletedFlag
NCx8x_00_Axis3Status_PresentPositionPresetAcknowledgedFlag 3327.07 BOOL  ; PresentPositionPresetAcknowledgedFlag
NCx8x_00_Axis3Status_RelativeMovementAcknowledgedFlag 3327.01 BOOL  ; RelativeMovementAcknowledgedFlag
NCx8x_00_Axis3Status_RelativeMovementFlag 3330.05 BOOL  ; RelativeMovementFlag
NCx8x_00_Axis3Status_ReverseJogging_InchingAcknowledgedFlag 3326.08 BOOL  ; ReverseJogging_InchingAcknowledgedFlag
NCx8x_00_Axis3Status_ReverseLimitInputFlag 3332.09 BOOL  ; ReverseLimitInputFlag
NCx8x_00_Axis3Status_ReverseTorqueLimitAcknowledgedFlag 3326.04 BOOL  ; ReverseTorqueLimitAcknowledgedFlag
NCx8x_00_Axis3Status_ReverseTorqueLimitOutputFlag 3332.04 BOOL  ; ReverseTorqueLimitOutputFlag
NCx8x_00_Axis3Status_SensorErrorFlag 3331.08 BOOL  ; SensorErrorFlag
NCx8x_00_Axis3Status_ServoDriveWarningFlag 3332.06 BOOL  ; ServoDriveWarningFlag
NCx8x_00_Axis3Status_ServoErrorFlag 3331.09 BOOL  ; ServoErrorFlag
NCx8x_00_Axis3Status_ServoLockAcknowledgedFlag 3326.00 BOOL  ; ServoLockAcknowledgedFlag
NCx8x_00_Axis3Status_ServoLockedFlag 3329.01 BOOL  ; ServoLockedFlag
NCx8x_00_Axis3Status_ServoONFlag 3332.00 BOOL  ; ServoONFlag
NCx8x_00_Axis3Status_ServoReadyFlag 3332.07 BOOL  ; ServoReadyFlag
NCx8x_00_Axis3Status_ServoUnlockAcknowledgedFlag 3326.15 BOOL  ; ServoUnlockAcknowledgedFlag
NCx8x_00_Axis3Status_ServoUnlockedFlag 3329.00 BOOL  ; ServoUnlockedFlag
NCx8x_00_Axis3Status_SpeedControlAcknowledgedFlag 3327.02 BOOL  ; SpeedControlAcknowledgedFlag
NCx8x_00_Axis3Status_SpeedControlFlag 3330.06 BOOL  ; SpeedControlFlag
NCx8x_00_Axis3Status_StartInvalidFlag 3328.08 BOOL  ; StartInvalidFlag
NCx8x_00_Axis3Status_StopExecutedFlag 3328.12 BOOL  ; StopExecutedFlag
NCx8x_00_Axis3Status_StopInputFlag 3328.04 BOOL  ; StopInputFlag
NCx8x_00_Axis3Status_StoppedatOriginFlag 3331.01 BOOL  ; StoppedatOriginFlag
NCx8x_00_Axis3Status_Zone0Flag 3331.13 BOOL  ; Zone0Flag
NCx8x_00_Axis3Status_Zone1Flag 3331.14 BOOL  ; Zone1Flag
NCx8x_00_Axis3Status_Zone2Flag 3331.15 BOOL  ; Zone2Flag
NCx8x_00_Axis4DirectOperation_DecelerationTime 3146 DINT  ; DecelerationTime
NCx8x_00_Axis4Status_AxisBusyFlag 3341.00 BOOL  ; AxisBusyFlag
NCx8x_00_Axis4Status_RelativeMovementFlag 3343.05 BOOL  ; RelativeMovementFlag
NCx8x_00_PCUControlInput_ABSEncoderBackupDataError 1513.05 BOOL  ; ABSEncoderBackupDataError
NCx8x_00_PCUControlInput_AllSlaveProcessDataCommunicationsFlag 1518.14 BOOL  ; AllSlaveProcessDataCommunicationsFlag
NCx8x_00_PCUControlInput_CommunicationsParameterSettingErrorFlag 1519.04 BOOL  ; CommunicationsParameterSettingErrorFlag
NCx8x_00_PCUControlInput_DataTransferCompletedFlag 1512.02 BOOL  ; DataTransferCompletedFlag
NCx8x_00_PCUControlInput_DataTransferFlag 1512.00 BOOL  ; DataTransferFlag
NCx8x_00_PCUControlInput_DataTransferInvalidFlag 1512.01 BOOL  ; DataTransferInvalidFlag
NCx8x_00_PCUControlInput_DownloadModeFlag 1512.10 BOOL  ; DownloadModeFlag
NCx8x_00_PCUControlInput_ErrorResetAcknowledgedFlag 1511.00 BOOL  ; ErrorResetAcknowledgedFlag
NCx8x_00_PCUControlInput_EtherCATDetectionProcessingFlag 1512.09 BOOL  ; EtherCATDetectionProcessingFlag
NCx8x_00_PCUControlInput_FatalProcessDataCommunicationsErrorFlag 1519.15 BOOL  ; FatalProcessDataCommunicationsErrorFlag
NCx8x_00_PCUControlInput_FrameSendTimingErrorFlag 1519.05 BOOL  ; FrameSendTimingErrorFlag
NCx8x_00_PCUControlInput_HardwareFailureFlag 1513.07 BOOL  ; HardwareFailureFlag
NCx8x_00_PCUControlInput_LinkOffErrorFlag 1519.09 BOOL  ; LinkOffErrorFlag
NCx8x_00_PCUControlInput_LinkStatusFlag 1518.13 BOOL  ; LinkStatusFlag
NCx8x_00_PCUControlInput_MemoryOperationAuxiliaryFlag0 1515.00 BOOL  ; MemoryOperationAuxiliaryFlag0
NCx8x_00_PCUControlInput_MemoryOperationAuxiliaryFlag1 1515.01 BOOL  ; MemoryOperationAuxiliaryFlag1
NCx8x_00_PCUControlInput_MemoryOperationAuxiliaryFlag10 1515.10 BOOL  ; MemoryOperationAuxiliaryFlag10
NCx8x_00_PCUControlInput_MemoryOperationAuxiliaryFlag11 1515.11 BOOL  ; MemoryOperationAuxiliaryFlag11
NCx8x_00_PCUControlInput_MemoryOperationAuxiliaryFlag12 1515.12 BOOL  ; MemoryOperationAuxiliaryFlag12
NCx8x_00_PCUControlInput_MemoryOperationAuxiliaryFlag13 1515.13 BOOL  ; MemoryOperationAuxiliaryFlag13
NCx8x_00_PCUControlInput_MemoryOperationAuxiliaryFlag14 1515.14 BOOL  ; MemoryOperationAuxiliaryFlag14
NCx8x_00_PCUControlInput_MemoryOperationAuxiliaryFlag15 1515.15 BOOL  ; MemoryOperationAuxiliaryFlag15
NCx8x_00_PCUControlInput_MemoryOperationAuxiliaryFlag2 1515.02 BOOL  ; MemoryOperationAuxiliaryFlag2
NCx8x_00_PCUControlInput_MemoryOperationAuxiliaryFlag3 1515.03 BOOL  ; MemoryOperationAuxiliaryFlag3
NCx8x_00_PCUControlInput_MemoryOperationAuxiliaryFlag4 1515.04 BOOL  ; MemoryOperationAuxiliaryFlag4
NCx8x_00_PCUControlInput_MemoryOperationAuxiliaryFlag5 1515.05 BOOL  ; MemoryOperationAuxiliaryFlag5
NCx8x_00_PCUControlInput_MemoryOperationAuxiliaryFlag6 1515.06 BOOL  ; MemoryOperationAuxiliaryFlag6
NCx8x_00_PCUControlInput_MemoryOperationAuxiliaryFlag7 1515.07 BOOL  ; MemoryOperationAuxiliaryFlag7
NCx8x_00_PCUControlInput_MemoryOperationAuxiliaryFlag8 1515.08 BOOL  ; MemoryOperationAuxiliaryFlag8
NCx8x_00_PCUControlInput_MemoryOperationAuxiliaryFlag9 1515.09 BOOL  ; MemoryOperationAuxiliaryFlag9
NCx8x_00_PCUControlInput_NetworkConfigurationErrorFlag 1519.01 BOOL  ; NetworkConfigurationErrorFlag
NCx8x_00_PCUControlInput_NetworkConfigurationVerificationErrorFlag 1519.00 BOOL  ; NetworkConfigurationVerificationErrorFlag
NCx8x_00_PCUControlInput_Node1CommunicationsErrorFlag 1524.00 BOOL  ; Node1CommunicationsErrorFlag
NCx8x_00_PCUControlInput_Node1MessageCommunicationsEnabledFlag 1522.00 BOOL  ; Node1MessageCommunicationsEnabledFlag
NCx8x_00_PCUControlInput_Node1NetworkParticipationFlag 1521.00 BOOL  ; Node1NetworkParticipationFlag
NCx8x_00_PCUControlInput_Node1NormalCommunicationsFlag 1523.00 BOOL  ; Node1NormalCommunicationsFlag
NCx8x_00_PCUControlInput_Node1RegisteredFlag 1520.00 BOOL  ; Node1RegisteredFlag
NCx8x_00_PCUControlInput_Node2CommunicationsErrorFlag 1524.01 BOOL  ; Node2CommunicationsErrorFlag
NCx8x_00_PCUControlInput_Node2MessageCommunicationsEnabledFlag 1522.01 BOOL  ; Node2MessageCommunicationsEnabledFlag
NCx8x_00_PCUControlInput_Node2NetworkParticipationFlag 1521.01 BOOL  ; Node2NetworkParticipationFlag
NCx8x_00_PCUControlInput_Node2NormalCommunicationsFlag 1523.01 BOOL  ; Node2NormalCommunicationsFlag
NCx8x_00_PCUControlInput_Node2RegisteredFlag 1520.01 BOOL  ; Node2RegisteredFlag
NCx8x_00_PCUControlInput_Node3CommunicationsErrorFlag 1524.02 BOOL  ; Node3CommunicationsErrorFlag
NCx8x_00_PCUControlInput_Node3MessageCommunicationsEnabledFlag 1522.02 BOOL  ; Node3MessageCommunicationsEnabledFlag
NCx8x_00_PCUControlInput_Node3NetworkParticipationFlag 1521.02 BOOL  ; Node3NetworkParticipationFlag
NCx8x_00_PCUControlInput_Node3NormalCommunicationsFlag 1523.02 BOOL  ; Node3NormalCommunicationsFlag
NCx8x_00_PCUControlInput_Node3RegisteredFlag 1520.02 BOOL  ; Node3RegisteredFlag
NCx8x_00_PCUControlInput_Node4CommunicationsErrorFlag 1524.03 BOOL  ; Node4CommunicationsErrorFlag
NCx8x_00_PCUControlInput_Node4MessageCommunicationsEnabledFlag 1522.03 BOOL  ; Node4MessageCommunicationsEnabledFlag
NCx8x_00_PCUControlInput_Node4NetworkParticipationFlag 1521.03 BOOL  ; Node4NetworkParticipationFlag
NCx8x_00_PCUControlInput_Node4NormalCommunicationsFlag 1523.03 BOOL  ; Node4NormalCommunicationsFlag
NCx8x_00_PCUControlInput_Node4RegisteredFlag 1520.03 BOOL  ; Node4RegisteredFlag
NCx8x_00_PCUControlInput_Node5CommunicationsErrorFlag 1524.04 BOOL  ; Node5CommunicationsErrorFlag
NCx8x_00_PCUControlInput_Node5MessageCommunicationsEnabledFlag 1522.04 BOOL  ; Node5MessageCommunicationsEnabledFlag
NCx8x_00_PCUControlInput_Node5NetworkParticipationFlag 1521.04 BOOL  ; Node5NetworkParticipationFlag
NCx8x_00_PCUControlInput_Node5NormalCommunicationsFlag 1523.04 BOOL  ; Node5NormalCommunicationsFlag
NCx8x_00_PCUControlInput_Node5RegisteredFlag 1520.04 BOOL  ; Node5RegisteredFlag
NCx8x_00_PCUControlInput_Node6CommunicationsErrorFlag 1524.05 BOOL  ; Node6CommunicationsErrorFlag
NCx8x_00_PCUControlInput_Node6MessageCommunicationsEnabledFlag 1522.05 BOOL  ; Node6MessageCommunicationsEnabledFlag
NCx8x_00_PCUControlInput_Node6NetworkParticipationFlag 1521.05 BOOL  ; Node6NetworkParticipationFlag
NCx8x_00_PCUControlInput_Node6NormalCommunicationsFlag 1523.05 BOOL  ; Node6NormalCommunicationsFlag
NCx8x_00_PCUControlInput_Node6RegisteredFlag 1520.05 BOOL  ; Node6RegisteredFlag
NCx8x_00_PCUControlInput_Node7CommunicationsErrorFlag 1524.06 BOOL  ; Node7CommunicationsErrorFlag
NCx8x_00_PCUControlInput_Node7MessageCommunicationsEnabledFlag 1522.06 BOOL  ; Node7MessageCommunicationsEnabledFlag
NCx8x_00_PCUControlInput_Node7NetworkParticipationFlag 1521.06 BOOL  ; Node7NetworkParticipationFlag
NCx8x_00_PCUControlInput_Node7NormalCommunicationsFlag 1523.06 BOOL  ; Node7NormalCommunicationsFlag
NCx8x_00_PCUControlInput_Node7RegisteredFlag 1520.06 BOOL  ; Node7RegisteredFlag
NCx8x_00_PCUControlInput_Node8CommunicationsErrorFlag 1524.07 BOOL  ; Node8CommunicationsErrorFlag
NCx8x_00_PCUControlInput_Node8MessageCommunicationsEnabledFlag 1522.07 BOOL  ; Node8MessageCommunicationsEnabledFlag
NCx8x_00_PCUControlInput_Node8NetworkParticipationFlag 1521.07 BOOL  ; Node8NetworkParticipationFlag
NCx8x_00_PCUControlInput_Node8NormalCommunicationsFlag 1523.07 BOOL  ; Node8NormalCommunicationsFlag
NCx8x_00_PCUControlInput_Node8RegisteredFlag 1520.07 BOOL  ; Node8RegisteredFlag
NCx8x_00_PCUControlInput_NonfatalProcessDataCommunicationsErrorFlag 1519.14 BOOL  ; NonfatalProcessDataCommunicationsErrorFlag
NCx8x_00_PCUControlInput_OverallAxisErrorFlag 1513.13 BOOL  ; OverallAxisErrorFlag
NCx8x_00_PCUControlInput_OverallErrorFlag 1513.15 BOOL  ; OverallErrorFlag
NCx8x_00_PCUControlInput_OverallMemoryOperationErrorFlag 1513.14 BOOL  ; OverallMemoryOperationErrorFlag
NCx8x_00_PCUControlInput_PCUErrorCode 1514 UINT  ; PCUErrorCode
NCx8x_00_PCUControlInput_PCUErrorFlag 1513.12 BOOL  ; PCUErrorFlag
NCx8x_00_PCUControlInput_PCUReadyFlag 1511.15 BOOL  ; PCUReadyFlag
NCx8x_00_PCUControlInput_PCUWarningFlag 1513.11 BOOL  ; PCUWarningFlag
NCx8x_00_PCUControlInput_PLCSystemErrorFlag 1513.09 BOOL  ; PLCSystemErrorFlag
NCx8x_00_PCUControlInput_ProcessDataCommunicationsErrorFlag 1519.02 BOOL  ; ProcessDataCommunicationsErrorFlag
NCx8x_00_PCUControlInput_ProcessDataReceptionTimeout 1519.03 BOOL  ; ProcessDataReceptionTimeout
NCx8x_00_PCUControlInput_ReadDataAcknowledgedFlag 1511.13 BOOL  ; ReadDataAcknowledgedFlag
NCx8x_00_PCUControlInput_ResettingErrorFlag 1512.04 BOOL  ; ResettingErrorFlag
NCx8x_00_PCUControlInput_RestoreErrorFlag 1513.00 BOOL  ; RestoreErrorFlag
NCx8x_00_PCUControlInput_SaveDataAcknowledgedFlag 1511.14 BOOL  ; SaveDataAcknowledgedFlag
NCx8x_00_PCUControlInput_SaveDataRequestFlag 1512.03 BOOL  ; SaveDataRequestFlag
NCx8x_00_PCUControlInput_SavedDataErrorFlag 1513.08 BOOL  ; SavedDataErrorFlag
NCx8x_00_PCUControlInput_SlaveALStatusErrorFlag 1519.12 BOOL  ; SlaveALStatusErrorFlag
NCx8x_00_PCUControlInput_SlaveInitializationErrorFlag 1519.11 BOOL  ; SlaveInitializationErrorFlag
NCx8x_00_PCUControlInput_SlaveNodeAddressDuplicatedFlag 1519.10 BOOL  ; SlaveNodeAddressDuplicatedFlag
NCx8x_00_PCUControlInput_TestModeFlag 1512.11 BOOL  ; TestModeFlag
NCx8x_00_PCUControlInput_WarningResetAcknowledgedFlag 1511.01 BOOL  ; WarningResetAcknowledgedFlag
NCx8x_00_PCUControlInput_WriteDataAckowledgeFlag 1511.12 BOOL  ; WriteDataAckowledgeFlag
NCx8x_00_PCUControlOutput_Axis1OriginProximityInputInternalMemoryArea 1507.00 BOOL  ; Axis1OriginProximityInputInternalMemoryArea
NCx8x_00_PCUControlOutput_Axis2OriginProximityInputInternalMemoryArea 1507.01 BOOL  ; Axis2OriginProximityInputInternalMemoryArea
NCx8x_00_PCUControlOutput_Axis3OriginProximityInputInternalMemoryArea 1507.02 BOOL  ; Axis3OriginProximityInputInternalMemoryArea
NCx8x_00_PCUControlOutput_Axis4OriginProximityInputInternalMemoryArea 1507.03 BOOL  ; Axis4OriginProximityInputInternalMemoryArea
NCx8x_00_PCUControlOutput_Axis5OriginProximityInputInternalMemoryArea 1507.04 BOOL  ; Axis5OriginProximityInputInternalMemoryArea
NCx8x_00_PCUControlOutput_Axis6OriginProximityInputInternalMemoryArea 1507.05 BOOL  ; Axis6OriginProximityInputInternalMemoryArea
NCx8x_00_PCUControlOutput_Axis7OriginProximityInputInternalMemoryArea 1507.06 BOOL  ; Axis7OriginProximityInputInternalMemoryArea
NCx8x_00_PCUControlOutput_Axis8OriginProximityInputInternalMemoryArea 1507.07 BOOL  ; Axis8OriginProximityInputInternalMemoryArea
NCx8x_00_PCUControlOutput_CPUUnitDataTransferAreaType 1502 UINT  ; CPUUnitDataTransferAreaType
NCx8x_00_PCUControlOutput_CPUUnitDataTransferStartWord 1503 UINT  ; CPUUnitDataTransferStartWord
NCx8x_00_PCUControlOutput_DataTransferWordsCount 1501 UINT  ; DataTransferWordsCount
NCx8x_00_PCUControlOutput_ErrorResetBit 1500.00 BOOL  ; ErrorResetBit
NCx8x_00_PCUControlOutput_PCUDataTransferArea 1504 UINT  ; PCUDataTransferArea
NCx8x_00_PCUControlOutput_PCUDataTransferBeginningWord1 1505 UINT  ; PCUDataTransferBeginningWord1
NCx8x_00_PCUControlOutput_PCUDataTransferBeginningWord2 1506 UINT  ; PCUDataTransferBeginningWord2
NCx8x_00_PCUControlOutput_PCUSetupBit 1500.15 BOOL  ; PCUSetupBit
NCx8x_00_PCUControlOutput_ReadDataBit 1500.13 BOOL  ; ReadDataBit
NCx8x_00_PCUControlOutput_SaveDataBit 1500.14 BOOL  ; SaveDataBit
NCx8x_00_PCUControlOutput_WarningResetBit 1500.01 BOOL  ; WarningResetBit
NCx8x_00_PCUControlOutput_WriteDataBit 1500.12 BOOL  ; WriteDataBit
NCx8x_00_Task1MemoryOperationStatus_ConditionInputWaitingFlag 3402.03 BOOL  ; ConditionInputWaitingFlag
NCx8x_00_Task1MemoryOperationStatus_DwellTimerWaitingFlag 3402.04 BOOL  ; DwellTimerWaitingFlag
NCx8x_00_Task1MemoryOperationStatus_ExecutingSequenceNumber 3404 UINT  ; ExecutingSequenceNumber
NCx8x_00_Task1MemoryOperationStatus_MCode 3405 UINT  ; MCode
NCx8x_00_Task1MemoryOperationStatus_MCodeResetAcknowledgedFlag 3400.04 BOOL  ; MCodeResetAcknowledgedFlag
NCx8x_00_Task1MemoryOperationStatus_MCodeResetWaitingFlag 3402.05 BOOL  ; MCodeResetWaitingFlag
NCx8x_00_Task1MemoryOperationStatus_MStrobeFlag 3402.06 BOOL  ; MStrobeFlag
NCx8x_00_Task1MemoryOperationStatus_MemoryOperationAxisOperationFlag 3402.02 BOOL  ; MemoryOperationAxisOperationFlag
NCx8x_00_Task1MemoryOperationStatus_MemoryOperationBusyFlag 3401.00 BOOL  ; MemoryOperationBusyFlag
NCx8x_00_Task1MemoryOperationStatus_MemoryOperationCompletedFlag 3401.13 BOOL  ; MemoryOperationCompletedFlag
NCx8x_00_Task1MemoryOperationStatus_MemoryOperationErrorCode 3403 UINT  ; MemoryOperationErrorCode
NCx8x_00_Task1MemoryOperationStatus_MemoryOperationErrorFlag 3402.12 BOOL  ; MemoryOperationErrorFlag
NCx8x_00_Task1MemoryOperationStatus_MemoryOperationExecutionErrorFlag 3402.10 BOOL  ; MemoryOperationExecutionErrorFlag
NCx8x_00_Task1MemoryOperationStatus_MemoryOperationIndependentStartAcknowledgedFlag 3400.02 BOOL  ; MemoryOperationIndependentStartAcknowledgedFlag
NCx8x_00_Task1MemoryOperationStatus_MemoryOperationStartAcknowledgedFlag 3400.01 BOOL  ; MemoryOperationStartAcknowledgedFlag
NCx8x_00_Task1MemoryOperationStatus_MemoryOperationStartEnabledFlag 3401.01 BOOL  ; MemoryOperationStartEnabledFlag
NCx8x_00_Task1MemoryOperationStatus_MemoryOperationStartInvalidFlag 3401.08 BOOL  ; MemoryOperationStartInvalidFlag
NCx8x_00_Task1MemoryOperationStatus_MemoryOperationStopAcknowledgedFlag 3400.15 BOOL  ; MemoryOperationStopAcknowledgedFlag
NCx8x_00_Task1MemoryOperationStatus_MemoryOperationStopExecutedFlag 3401.12 BOOL  ; MemoryOperationStopExecutedFlag
NCx8x_00_Task1MemoryOperationStatus_MemoryOperationStopInputFlag 3401.04 BOOL  ; MemoryOperationStopInputFlag
NCx8x_00_Task1MemoryOperationStatus_MemoryOperationStoppedFlag 3402.00 BOOL  ; MemoryOperationStoppedFlag
NCx8x_00_Task1MemoryOperationStatus_MemoryOperationWaitingFlag 3402.01 BOOL  ; MemoryOperationWaitingFlag
NCx8x_00_Task1MemoryOperationStatus_MemoryOperationWarningFlag 3402.11 BOOL  ; MemoryOperationWarningFlag
NCx8x_00_Task1MemoryOperationStatus_SequenceNumberEnableAcknowledgedFlag 3400.00 BOOL  ; SequenceNumberEnableAcknowledgedFlag
NCx8x_00_Task1MemoryOperationStatus_TeachingAcknowledgedFlag 3400.05 BOOL  ; TeachingAcknowledgedFlag
NCx8x_00_Task1MemoryOperationStatus_TeachingCompletedFlag 3401.14 BOOL  ; TeachingCompletedFlag
NCx8x_00_Task1MemoryOperationStatus_TeachingInvalidFlag 3401.09 BOOL  ; TeachingInvalidFlag
NCx8x_00_Task1MemoryOperation_MCodeResetBit 3200.04 BOOL  ; MCodeResetBit
NCx8x_00_Task1MemoryOperation_MemoryOperationIndependentStartBit 3200.02 BOOL  ; MemoryOperationIndependentStartBit
NCx8x_00_Task1MemoryOperation_MemoryOperationStartBit 3200.01 BOOL  ; MemoryOperationStartBit
NCx8x_00_Task1MemoryOperation_MemoryOperationStopBit 3200.15 BOOL  ; MemoryOperationStopBit
NCx8x_00_Task1MemoryOperation_SequenceNumber 3201 UINT  ; SequenceNumber
NCx8x_00_Task1MemoryOperation_SequenceNumberEnableBit 3200.00 BOOL  ; SequenceNumberEnableBit
NCx8x_00_Task1MemoryOperation_TeachingAddress 3202 UINT  ; TeachingAddress
NCx8x_00_Task1MemoryOperation_TeachingBit 3200.05 BOOL  ; TeachingBit
NCx8x_00_Task2MemoryOperationStatus_ConditionInputWaitingFlag 3408.03 BOOL  ; ConditionInputWaitingFlag
NCx8x_00_Task2MemoryOperationStatus_DwellTimerWaitingFlag 3408.04 BOOL  ; DwellTimerWaitingFlag
NCx8x_00_Task2MemoryOperationStatus_ExecutingSequenceNumber 3410 UINT  ; ExecutingSequenceNumber
NCx8x_00_Task2MemoryOperationStatus_MCode 3411 UINT  ; MCode
NCx8x_00_Task2MemoryOperationStatus_MCodeResetAcknowledgedFlag 3406.04 BOOL  ; MCodeResetAcknowledgedFlag
NCx8x_00_Task2MemoryOperationStatus_MCodeResetWaitingFlag 3408.05 BOOL  ; MCodeResetWaitingFlag
NCx8x_00_Task2MemoryOperationStatus_MStrobeFlag 3408.06 BOOL  ; MStrobeFlag
NCx8x_00_Task2MemoryOperationStatus_MemoryOperationAxisOperationFlag 3408.02 BOOL  ; MemoryOperationAxisOperationFlag
NCx8x_00_Task2MemoryOperationStatus_MemoryOperationBusyFlag 3407.00 BOOL  ; MemoryOperationBusyFlag
NCx8x_00_Task2MemoryOperationStatus_MemoryOperationCompletedFlag 3407.13 BOOL  ; MemoryOperationCompletedFlag
NCx8x_00_Task2MemoryOperationStatus_MemoryOperationErrorCode 3409 UINT  ; MemoryOperationErrorCode
NCx8x_00_Task2MemoryOperationStatus_MemoryOperationErrorFlag 3408.12 BOOL  ; MemoryOperationErrorFlag
NCx8x_00_Task2MemoryOperationStatus_MemoryOperationExecutionErrorFlag 3408.10 BOOL  ; MemoryOperationExecutionErrorFlag
NCx8x_00_Task2MemoryOperationStatus_MemoryOperationIndependentStartAcknowledgedFlag 3406.02 BOOL  ; MemoryOperationIndependentStartAcknowledgedFlag
NCx8x_00_Task2MemoryOperationStatus_MemoryOperationStartAcknowledgedFlag 3406.01 BOOL  ; MemoryOperationStartAcknowledgedFlag
NCx8x_00_Task2MemoryOperationStatus_MemoryOperationStartEnabledFlag 3407.01 BOOL  ; MemoryOperationStartEnabledFlag
NCx8x_00_Task2MemoryOperationStatus_MemoryOperationStartInvalidFlag 3407.08 BOOL  ; MemoryOperationStartInvalidFlag
NCx8x_00_Task2MemoryOperationStatus_MemoryOperationStopAcknowledgedFlag 3406.15 BOOL  ; MemoryOperationStopAcknowledgedFlag
NCx8x_00_Task2MemoryOperationStatus_MemoryOperationStopExecutedFlag 3407.12 BOOL  ; MemoryOperationStopExecutedFlag
NCx8x_00_Task2MemoryOperationStatus_MemoryOperationStopInputFlag 3407.04 BOOL  ; MemoryOperationStopInputFlag
NCx8x_00_Task2MemoryOperationStatus_MemoryOperationStoppedFlag 3408.00 BOOL  ; MemoryOperationStoppedFlag
NCx8x_00_Task2MemoryOperationStatus_MemoryOperationWaitingFlag 3408.01 BOOL  ; MemoryOperationWaitingFlag
NCx8x_00_Task2MemoryOperationStatus_MemoryOperationWarningFlag 3408.11 BOOL  ; MemoryOperationWarningFlag
NCx8x_00_Task2MemoryOperationStatus_SequenceNumberEnableAcknowledgedFlag 3406.00 BOOL  ; SequenceNumberEnableAcknowledgedFlag
NCx8x_00_Task2MemoryOperationStatus_TeachingAcknowledgedFlag 3406.05 BOOL  ; TeachingAcknowledgedFlag
NCx8x_00_Task2MemoryOperationStatus_TeachingCompletedFlag 3407.14 BOOL  ; TeachingCompletedFlag
NCx8x_00_Task2MemoryOperationStatus_TeachingInvalidFlag 3407.09 BOOL  ; TeachingInvalidFlag
NCx8x_00_Task2MemoryOperation_MCodeResetBit 3203.04 BOOL  ; MCodeResetBit
NCx8x_00_Task2MemoryOperation_MemoryOperationIndependentStartBit 3203.02 BOOL  ; MemoryOperationIndependentStartBit
NCx8x_00_Task2MemoryOperation_MemoryOperationStartBit 3203.01 BOOL  ; MemoryOperationStartBit
NCx8x_00_Task2MemoryOperation_MemoryOperationStopBit 3203.15 BOOL  ; MemoryOperationStopBit
NCx8x_00_Task2MemoryOperation_SequenceNumber 3204 UINT  ; SequenceNumber
NCx8x_00_Task2MemoryOperation_SequenceNumberEnableBit 3203.00 BOOL  ; SequenceNumberEnableBit
NCx8x_00_Task2MemoryOperation_TeachingAddress 3205 UINT  ; TeachingAddress
NCx8x_00_Task2MemoryOperation_TeachingBit 3203.05 BOOL  ; TeachingBit
NCx8x_00_Task3MemoryOperationStatus_ConditionInputWaitingFlag 3414.03 BOOL  ; ConditionInputWaitingFlag
NCx8x_00_Task3MemoryOperationStatus_DwellTimerWaitingFlag 3414.04 BOOL  ; DwellTimerWaitingFlag
NCx8x_00_Task3MemoryOperationStatus_ExecutingSequenceNumber 3416 UINT  ; ExecutingSequenceNumber
NCx8x_00_Task3MemoryOperationStatus_MCode 3417 UINT  ; MCode
NCx8x_00_Task3MemoryOperationStatus_MCodeResetAcknowledgedFlag 3412.04 BOOL  ; MCodeResetAcknowledgedFlag
NCx8x_00_Task3MemoryOperationStatus_MCodeResetWaitingFlag 3414.05 BOOL  ; MCodeResetWaitingFlag
NCx8x_00_Task3MemoryOperationStatus_MStrobeFlag 3414.06 BOOL  ; MStrobeFlag
NCx8x_00_Task3MemoryOperationStatus_MemoryOperationAxisOperationFlag 3414.02 BOOL  ; MemoryOperationAxisOperationFlag
NCx8x_00_Task3MemoryOperationStatus_MemoryOperationBusyFlag 3413.00 BOOL  ; MemoryOperationBusyFlag
NCx8x_00_Task3MemoryOperationStatus_MemoryOperationCompletedFlag 3413.13 BOOL  ; MemoryOperationCompletedFlag
NCx8x_00_Task3MemoryOperationStatus_MemoryOperationErrorCode 3415 UINT  ; MemoryOperationErrorCode
NCx8x_00_Task3MemoryOperationStatus_MemoryOperationErrorFlag 3414.12 BOOL  ; MemoryOperationErrorFlag
NCx8x_00_Task3MemoryOperationStatus_MemoryOperationExecutionErrorFlag 3414.10 BOOL  ; MemoryOperationExecutionErrorFlag
NCx8x_00_Task3MemoryOperationStatus_MemoryOperationIndependentStartAcknowledgedFlag 3412.02 BOOL  ; MemoryOperationIndependentStartAcknowledgedFlag
NCx8x_00_Task3MemoryOperationStatus_MemoryOperationStartAcknowledgedFlag 3412.01 BOOL  ; MemoryOperationStartAcknowledgedFlag
NCx8x_00_Task3MemoryOperationStatus_MemoryOperationStartEnabledFlag 3413.01 BOOL  ; MemoryOperationStartEnabledFlag
NCx8x_00_Task3MemoryOperationStatus_MemoryOperationStartInvalidFlag 3413.08 BOOL  ; MemoryOperationStartInvalidFlag
NCx8x_00_Task3MemoryOperationStatus_MemoryOperationStopAcknowledgedFlag 3412.15 BOOL  ; MemoryOperationStopAcknowledgedFlag
NCx8x_00_Task3MemoryOperationStatus_MemoryOperationStopExecutedFlag 3413.12 BOOL  ; MemoryOperationStopExecutedFlag
NCx8x_00_Task3MemoryOperationStatus_MemoryOperationStopInputFlag 3413.04 BOOL  ; MemoryOperationStopInputFlag
NCx8x_00_Task3MemoryOperationStatus_MemoryOperationStoppedFlag 3414.00 BOOL  ; MemoryOperationStoppedFlag
NCx8x_00_Task3MemoryOperationStatus_MemoryOperationWaitingFlag 3414.01 BOOL  ; MemoryOperationWaitingFlag
NCx8x_00_Task3MemoryOperationStatus_MemoryOperationWarningFlag 3414.11 BOOL  ; MemoryOperationWarningFlag
NCx8x_00_Task3MemoryOperationStatus_SequenceNumberEnableAcknowledgedFlag 3412.00 BOOL  ; SequenceNumberEnableAcknowledgedFlag
NCx8x_00_Task3MemoryOperationStatus_TeachingAcknowledgedFlag 3412.05 BOOL  ; TeachingAcknowledgedFlag
NCx8x_00_Task3MemoryOperationStatus_TeachingCompletedFlag 3413.14 BOOL  ; TeachingCompletedFlag
NCx8x_00_Task3MemoryOperationStatus_TeachingInvalidFlag 3413.09 BOOL  ; TeachingInvalidFlag
NCx8x_00_Task3MemoryOperation_MCodeResetBit 3206.04 BOOL  ; MCodeResetBit
NCx8x_00_Task3MemoryOperation_MemoryOperationIndependentStartBit 3206.02 BOOL  ; MemoryOperationIndependentStartBit
NCx8x_00_Task3MemoryOperation_MemoryOperationStartBit 3206.01 BOOL  ; MemoryOperationStartBit
NCx8x_00_Task3MemoryOperation_MemoryOperationStopBit 3206.15 BOOL  ; MemoryOperationStopBit
NCx8x_00_Task3MemoryOperation_SequenceNumber 3207 UINT  ; SequenceNumber
NCx8x_00_Task3MemoryOperation_SequenceNumberEnableBit 3206.00 BOOL  ; SequenceNumberEnableBit
NCx8x_00_Task3MemoryOperation_TeachingAddress 3208 UINT  ; TeachingAddress
NCx8x_00_Task3MemoryOperation_TeachingBit 3206.05 BOOL  ; TeachingBit
NCx8x_00_Task4MemoryOperationStatus_ConditionInputWaitingFlag 3420.03 BOOL  ; ConditionInputWaitingFlag
NCx8x_00_Task4MemoryOperationStatus_DwellTimerWaitingFlag 3420.04 BOOL  ; DwellTimerWaitingFlag
NCx8x_00_Task4MemoryOperationStatus_ExecutingSequenceNumber 3422 UINT  ; ExecutingSequenceNumber
NCx8x_00_Task4MemoryOperationStatus_MCode 3423 UINT  ; MCode
NCx8x_00_Task4MemoryOperationStatus_MCodeResetAcknowledgedFlag 3418.04 BOOL  ; MCodeResetAcknowledgedFlag
NCx8x_00_Task4MemoryOperationStatus_MCodeResetWaitingFlag 3420.05 BOOL  ; MCodeResetWaitingFlag
NCx8x_00_Task4MemoryOperationStatus_MStrobeFlag 3420.06 BOOL  ; MStrobeFlag
NCx8x_00_Task4MemoryOperationStatus_MemoryOperationAxisOperationFlag 3420.02 BOOL  ; MemoryOperationAxisOperationFlag
NCx8x_00_Task4MemoryOperationStatus_MemoryOperationBusyFlag 3419.00 BOOL  ; MemoryOperationBusyFlag
NCx8x_00_Task4MemoryOperationStatus_MemoryOperationCompletedFlag 3419.13 BOOL  ; MemoryOperationCompletedFlag
NCx8x_00_Task4MemoryOperationStatus_MemoryOperationErrorCode 3421 UINT  ; MemoryOperationErrorCode
NCx8x_00_Task4MemoryOperationStatus_MemoryOperationErrorFlag 3420.12 BOOL  ; MemoryOperationErrorFlag
NCx8x_00_Task4MemoryOperationStatus_MemoryOperationExecutionErrorFlag 3420.10 BOOL  ; MemoryOperationExecutionErrorFlag
NCx8x_00_Task4MemoryOperationStatus_MemoryOperationIndependentStartAcknowledgedFlag 3418.02 BOOL  ; MemoryOperationIndependentStartAcknowledgedFlag
NCx8x_00_Task4MemoryOperationStatus_MemoryOperationStartAcknowledgedFlag 3418.01 BOOL  ; MemoryOperationStartAcknowledgedFlag
NCx8x_00_Task4MemoryOperationStatus_MemoryOperationStartEnabledFlag 3419.01 BOOL  ; MemoryOperationStartEnabledFlag
NCx8x_00_Task4MemoryOperationStatus_MemoryOperationStartInvalidFlag 3419.08 BOOL  ; MemoryOperationStartInvalidFlag
NCx8x_00_Task4MemoryOperationStatus_MemoryOperationStopAcknowledgedFlag 3418.15 BOOL  ; MemoryOperationStopAcknowledgedFlag
NCx8x_00_Task4MemoryOperationStatus_MemoryOperationStopExecutedFlag 3419.12 BOOL  ; MemoryOperationStopExecutedFlag
NCx8x_00_Task4MemoryOperationStatus_MemoryOperationStopInputFlag 3419.04 BOOL  ; MemoryOperationStopInputFlag
NCx8x_00_Task4MemoryOperationStatus_MemoryOperationStoppedFlag 3420.00 BOOL  ; MemoryOperationStoppedFlag
NCx8x_00_Task4MemoryOperationStatus_MemoryOperationWaitingFlag 3420.01 BOOL  ; MemoryOperationWaitingFlag
NCx8x_00_Task4MemoryOperationStatus_MemoryOperationWarningFlag 3420.11 BOOL  ; MemoryOperationWarningFlag
NCx8x_00_Task4MemoryOperationStatus_SequenceNumberEnableAcknowledgedFlag 3418.00 BOOL  ; SequenceNumberEnableAcknowledgedFlag
NCx8x_00_Task4MemoryOperationStatus_TeachingAcknowledgedFlag 3418.05 BOOL  ; TeachingAcknowledgedFlag
NCx8x_00_Task4MemoryOperationStatus_TeachingCompletedFlag 3419.14 BOOL  ; TeachingCompletedFlag
NCx8x_00_Task4MemoryOperationStatus_TeachingInvalidFlag 3419.09 BOOL  ; TeachingInvalidFlag
NCx8x_00_Task4MemoryOperation_MCodeResetBit 3209.04 BOOL  ; MCodeResetBit
NCx8x_00_Task4MemoryOperation_MemoryOperationIndependentStartBit 3209.02 BOOL  ; MemoryOperationIndependentStartBit
NCx8x_00_Task4MemoryOperation_MemoryOperationStartBit 3209.01 BOOL  ; MemoryOperationStartBit
NCx8x_00_Task4MemoryOperation_MemoryOperationStopBit 3209.15 BOOL  ; MemoryOperationStopBit
NCx8x_00_Task4MemoryOperation_SequenceNumber 3210 UINT  ; SequenceNumber
NCx8x_00_Task4MemoryOperation_SequenceNumberEnableBit 3209.00 BOOL  ; SequenceNumberEnableBit
NCx8x_00_Task4MemoryOperation_TeachingAddress 3211 UINT  ; TeachingAddress
NCx8x_00_Task4MemoryOperation_TeachingBit 3209.05 BOOL  ; TeachingBit
Posicao_Corte_Inicial D1010 DINT  ; Posição nipe
Preset_Reb_Inf D102 REAL  ; Valor desejado de saida para o Rebobinador inferior
Preset_Reb_Sup D100 REAL  ; Valor para saída analógica
Pulso_Inicializacao W2.00 BOOL
Rebobinador_Inf Escala_SA
Rebobinador_Inf2 Escala_SA
Rebobinador_Sup Escala_SA
Rebobinador_sup2 Escala_SA
Relacao_TRO Relacao_motor
Reset W2.01 BOOL  ; Reset inicialização
SP_Saida_1_Aquec 2010 CHANNEL  ; Setpoint da saída de aquecimento 1
SP_Saida_2_Aquec 2011 CHANNEL  ; Setpoint da saída de aquecimento 2
SP_Saida_3_Aquec 2020 CHANNEL  ; Setpoint da saída de aquecimento 3
SP_Saida_4_Aquec 2021 CHANNEL  ; Setpoint da saída de aquecimento 4
S_LOCK_SERVO_REB_INF 1.14 BOOL  ; Saída Habilita servo Rebobinador inferior 1
S_LOCK_SERVO_REB_SUP 1.15 BOOL  ; Saída Habilita servo Rebobinador superior 1
S_MARCADOR 1.03 BOOL  ; Saída para etiquetador
S_NIP 1.00 BOOL  ; tracionador NIP
S_NIP_SEL 1.02 BOOL  ; Tracionador Nip Selagem
S_ROLDANA_SEL 1.04 BOOL
S_SEL 1.01 BOOL  ; Tracionador Selagem
Saida_Analógica_1 Escala_SA
Vel_Nipe Calc_Vel
Vel_Selagem Calc_Vel
Vel_TRO Calc_Vel_TRO
ZONA1 _TCx004_ExecuteAT
ZONA2 _TCx004_ExecuteAT
ZONA3 _TCx004_ExecuteAT
ZONA4 _TCx004_ExecuteAT
ZONA5 _TCx004_ExecuteAT

## Program NewProgram1 (cyclic task 0)
Local symbols
CONTAGEM_PAR D672 CHANNEL
aux_preset_rebobinador REAL

### Section TRO

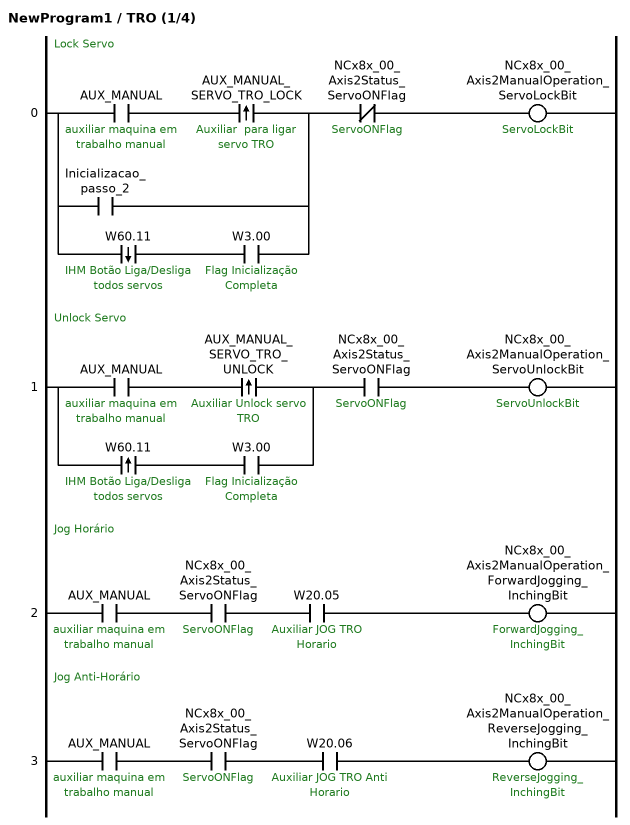
; rung 0: Lock Servo
LD AUX_MANUAL  ; auxiliar maquina em trabalho manual
@AND AUX_MANUAL_SERVO_TRO_LOCK  ; Auxiliar  para ligar servo TRO
OR Inicializacao_passo_2
%LD W60.11  ; IHM Botão Liga/Desliga todos servos
AND W3.00  ; Flag Inicialização Completa
ORLD
ANDNOT NCx8x_00_Axis2Status_ServoONFlag  ; ServoONFlag
OUT NCx8x_00_Axis2ManualOperation_ServoLockBit  ; ServoLockBit
; rung 1: Unlock Servo
LD AUX_MANUAL  ; auxiliar maquina em trabalho manual
@AND AUX_MANUAL_SERVO_TRO_UNLOCK  ; Auxiliar Unlock servo TRO
@LD W60.11  ; IHM Botão Liga/Desliga todos servos
AND W3.00  ; Flag Inicialização Completa
ORLD
AND NCx8x_00_Axis2Status_ServoONFlag  ; ServoONFlag
OUT NCx8x_00_Axis2ManualOperation_ServoUnlockBit  ; ServoUnlockBit
; rung 2: Jog Horário
LD AUX_MANUAL  ; auxiliar maquina em trabalho manual
AND NCx8x_00_Axis2Status_ServoONFlag  ; ServoONFlag
AND W20.05  ; Auxiliar JOG TRO Horario
OUT NCx8x_00_Axis2ManualOperation_ForwardJogging_InchingBit  ; ForwardJogging_InchingBit
; rung 3: Jog Anti-Horário
LD AUX_MANUAL  ; auxiliar maquina em trabalho manual
AND NCx8x_00_Axis2Status_ServoONFlag  ; ServoONFlag
AND W20.06  ; Auxiliar JOG TRO Anti Horario
OUT NCx8x_00_Axis2ManualOperation_ReverseJogging_InchingBit  ; ReverseJogging_InchingBit

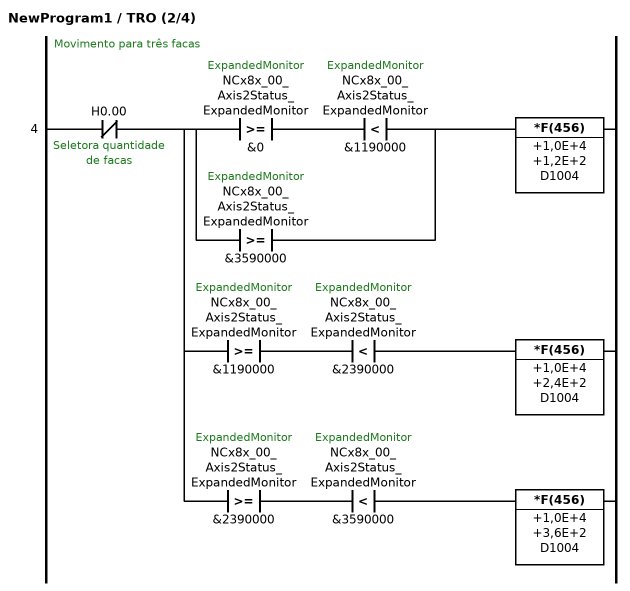
; rung 4: Movimento para três facas
LDNOT H0.00  ; Seletora quantidade de facas
OUT TR0
LD>=L(326) NCx8x_00_Axis2Status_ExpandedMonitor &0  ; ExpandedMonitor
AND<L(311) NCx8x_00_Axis2Status_ExpandedMonitor &1190000  ; ExpandedMonitor
OR>=L(326) NCx8x_00_Axis2Status_ExpandedMonitor &3590000  ; ExpandedMonitor
ANDLD
*F(456) +1,0E+4 +1,2E+2 D1004
LD TR0
AND>=L(326) NCx8x_00_Axis2Status_ExpandedMonitor &1190000  ; ExpandedMonitor
AND<L(311) NCx8x_00_Axis2Status_ExpandedMonitor &2390000  ; ExpandedMonitor
*F(456) +1,0E+4 +2,4E+2 D1004
LD TR0
AND>=L(326) NCx8x_00_Axis2Status_ExpandedMonitor &2390000  ; ExpandedMonitor
AND<L(311) NCx8x_00_Axis2Status_ExpandedMonitor &3590000  ; ExpandedMonitor
*F(456) +1,0E+4 +3,6E+2 D1004

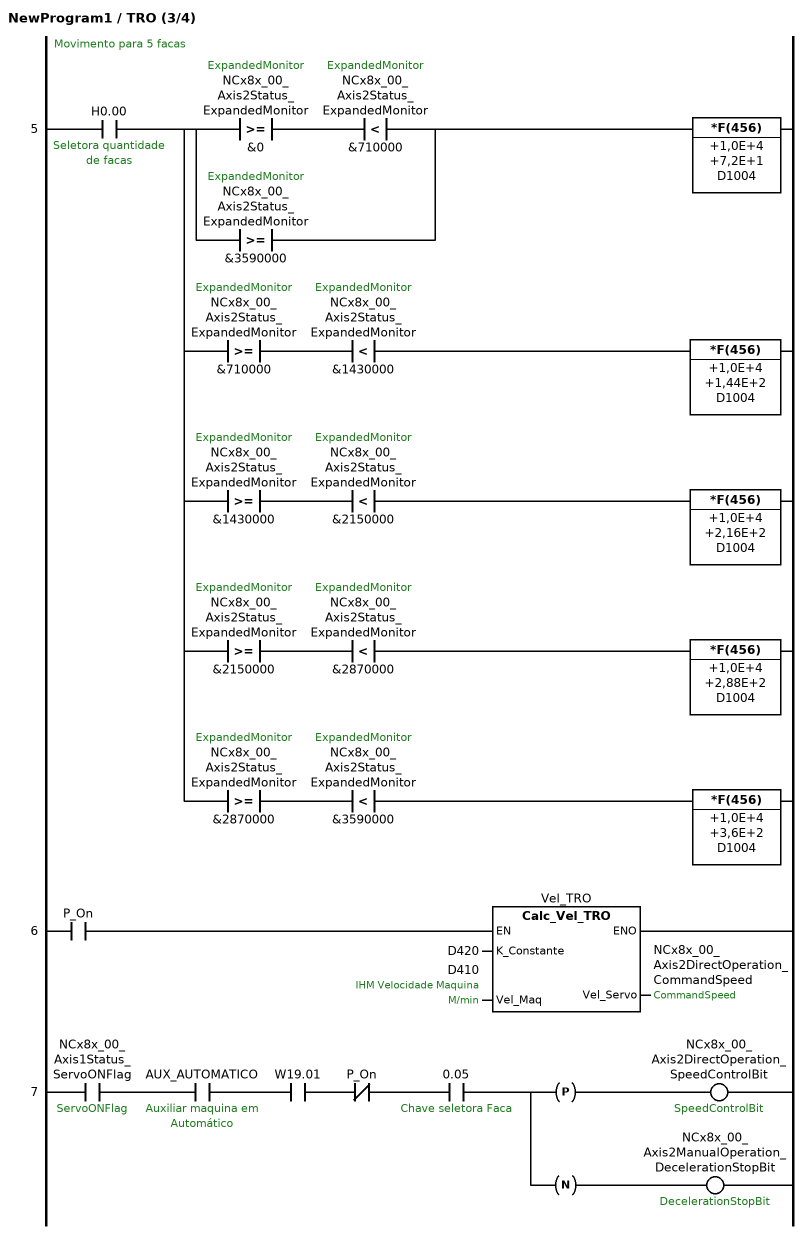
; rung 5: Movimento para 5 facas
LD H0.00  ; Seletora quantidade de facas
OUT TR0
LD>=L(326) NCx8x_00_Axis2Status_ExpandedMonitor &0  ; ExpandedMonitor
AND<L(311) NCx8x_00_Axis2Status_ExpandedMonitor &710000  ; ExpandedMonitor
OR>=L(326) NCx8x_00_Axis2Status_ExpandedMonitor &3590000  ; ExpandedMonitor
ANDLD
*F(456) +1,0E+4 +7,2E+1 D1004
LD TR0
AND>=L(326) NCx8x_00_Axis2Status_ExpandedMonitor &710000  ; ExpandedMonitor
AND<L(311) NCx8x_00_Axis2Status_ExpandedMonitor &1430000  ; ExpandedMonitor
*F(456) +1,0E+4 +1,44E+2 D1004
LD TR0
AND>=L(326) NCx8x_00_Axis2Status_ExpandedMonitor &1430000  ; ExpandedMonitor
AND<L(311) NCx8x_00_Axis2Status_ExpandedMonitor &2150000  ; ExpandedMonitor
*F(456) +1,0E+4 +2,16E+2 D1004
LD TR0
AND>=L(326) NCx8x_00_Axis2Status_ExpandedMonitor &2150000  ; ExpandedMonitor
AND<L(311) NCx8x_00_Axis2Status_ExpandedMonitor &2870000  ; ExpandedMonitor
*F(456) +1,0E+4 +2,88E+2 D1004
LD TR0
AND>=L(326) NCx8x_00_Axis2Status_ExpandedMonitor &2870000  ; ExpandedMonitor
AND<L(311) NCx8x_00_Axis2Status_ExpandedMonitor &3590000  ; ExpandedMonitor
*F(456) +1,0E+4 +3,6E+2 D1004
; rung 6
LD P_On
CALL Vel_TRO : Calc_Vel_TRO (K_Constante := D420, Vel_Maq := D410, Vel_Servo => NCx8x_00_Axis2DirectOperation_CommandSpeed)  ; IHM Velocidade Maquina M/min, CommandSpeed
; rung 7
LD NCx8x_00_Axis1Status_ServoONFlag  ; ServoONFlag
AND AUX_AUTOMATICO  ; Auxiliar maquina em Automático
AND W19.01
ANDNOT P_On
AND 0.05  ; Chave seletora Faca
OUT TR0
UP(521)
OUT NCx8x_00_Axis2DirectOperation_SpeedControlBit  ; SpeedControlBit
LD TR0
DOWN(522)
OUT NCx8x_00_Axis2ManualOperation_DecelerationStopBit  ; DecelerationStopBit

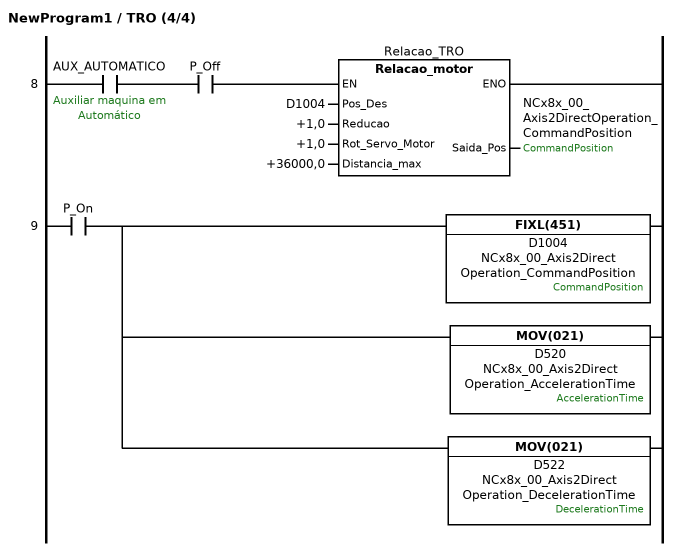
; rung 8
LD AUX_AUTOMATICO  ; Auxiliar maquina em Automático
AND P_Off
CALL Relacao_TRO : Relacao_motor (Pos_Des := D1004, Reducao := +1,0, Rot_Servo_Motor := +1,0, Distancia_max := +36000,0, Saida_Pos => NCx8x_00_Axis2DirectOperation_CommandPosition)  ; CommandPosition
; rung 9
LD P_On
FIXL(451) D1004 NCx8x_00_Axis2DirectOperation_CommandPosition  ; CommandPosition
MOV(021) D520 NCx8x_00_Axis2DirectOperation_AccelerationTime  ; AccelerationTime
MOV(021) D522 NCx8x_00_Axis2DirectOperation_DecelerationTime  ; DecelerationTime

### Section NIP

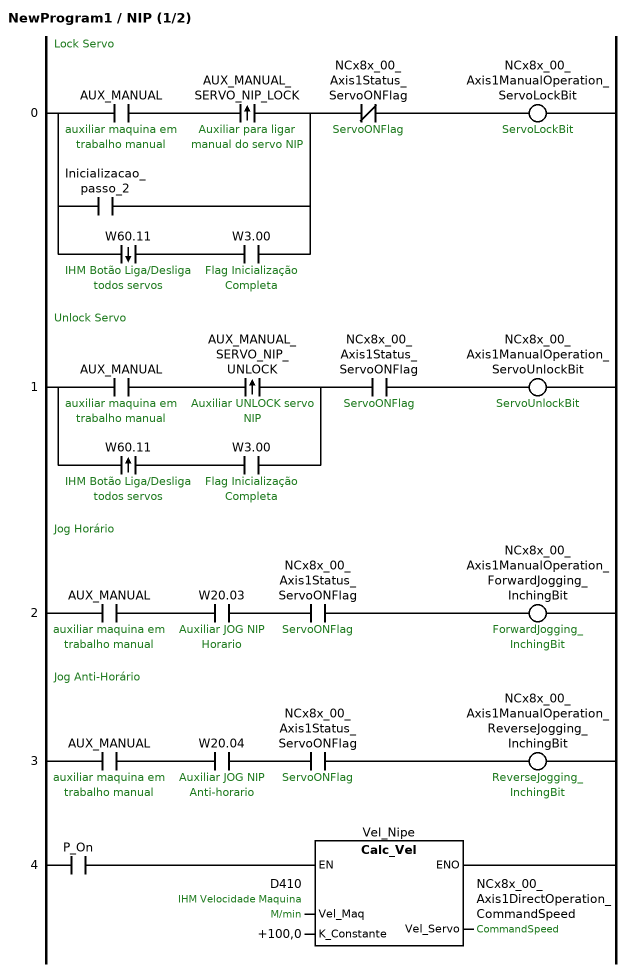
; rung 0: Lock Servo
LD AUX_MANUAL  ; auxiliar maquina em trabalho manual
@AND AUX_MANUAL_SERVO_NIP_LOCK  ; Auxiliar para ligar manual do servo NIP
OR Inicializacao_passo_2
%LD W60.11  ; IHM Botão Liga/Desliga todos servos
AND W3.00  ; Flag Inicialização Completa
ORLD
ANDNOT NCx8x_00_Axis1Status_ServoONFlag  ; ServoONFlag
OUT NCx8x_00_Axis1ManualOperation_ServoLockBit  ; ServoLockBit
; rung 1: Unlock Servo
LD AUX_MANUAL  ; auxiliar maquina em trabalho manual
@AND AUX_MANUAL_SERVO_NIP_UNLOCK  ; Auxiliar UNLOCK servo NIP
@LD W60.11  ; IHM Botão Liga/Desliga todos servos
AND W3.00  ; Flag Inicialização Completa
ORLD
AND NCx8x_00_Axis1Status_ServoONFlag  ; ServoONFlag
OUT NCx8x_00_Axis1ManualOperation_ServoUnlockBit  ; ServoUnlockBit
; rung 2: Jog Horário
LD AUX_MANUAL  ; auxiliar maquina em trabalho manual
AND W20.03  ; Auxiliar JOG NIP Horario
AND NCx8x_00_Axis1Status_ServoONFlag  ; ServoONFlag
OUT NCx8x_00_Axis1ManualOperation_ForwardJogging_InchingBit  ; ForwardJogging_InchingBit
; rung 3: Jog Anti-Horário
LD AUX_MANUAL  ; auxiliar maquina em trabalho manual
AND W20.04  ; Auxiliar JOG NIP Anti-horario
AND NCx8x_00_Axis1Status_ServoONFlag  ; ServoONFlag
OUT NCx8x_00_Axis1ManualOperation_ReverseJogging_InchingBit  ; ReverseJogging_InchingBit
; rung 4
LD P_On
CALL Vel_Nipe : Calc_Vel (Vel_Maq := D410, K_Constante := +100,0, Vel_Servo => NCx8x_00_Axis1DirectOperation_CommandSpeed)  ; IHM Velocidade Maquina M/min, CommandSpeed

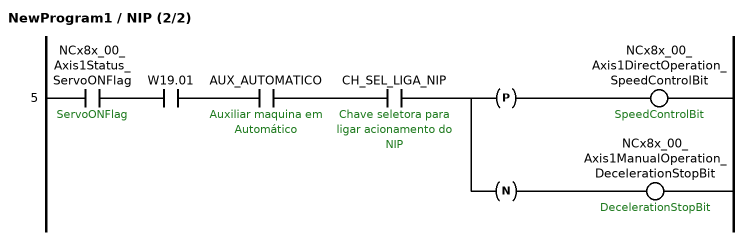
; rung 5
LD NCx8x_00_Axis1Status_ServoONFlag  ; ServoONFlag
AND W19.01
AND AUX_AUTOMATICO  ; Auxiliar maquina em Automático
AND CH_SEL_LIGA_NIP  ; Chave seletora para ligar acionamento do NIP
OUT TR0
UP(521)
OUT NCx8x_00_Axis1DirectOperation_SpeedControlBit  ; SpeedControlBit
LD TR0
DOWN(522)
OUT NCx8x_00_Axis1ManualOperation_DecelerationStopBit  ; DecelerationStopBit

### Section SEL

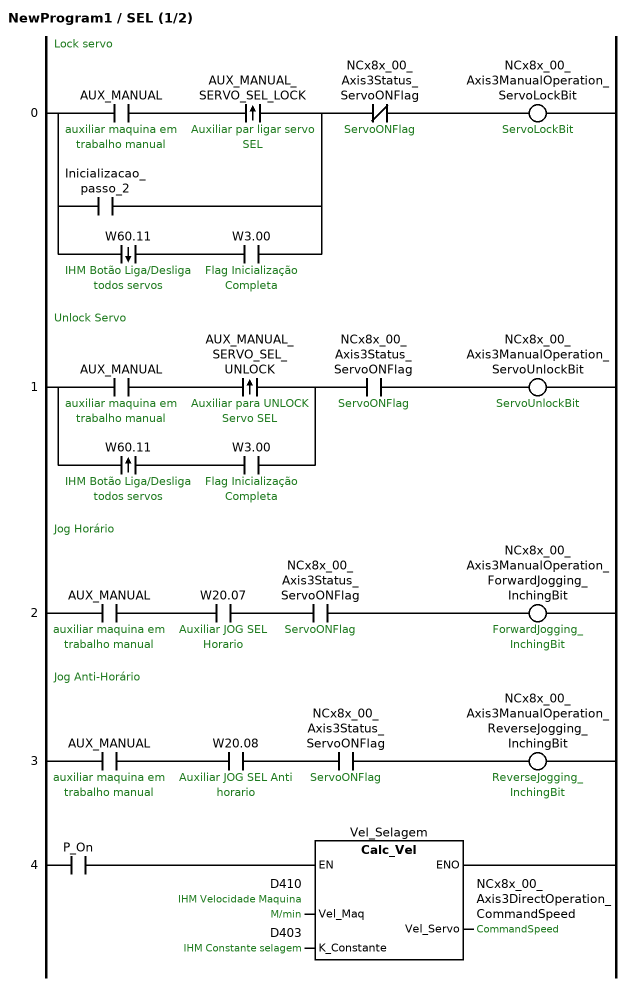
; rung 0: Lock servo
LD AUX_MANUAL  ; auxiliar maquina em trabalho manual
@AND AUX_MANUAL_SERVO_SEL_LOCK  ; Auxiliar par ligar servo SEL
OR Inicializacao_passo_2
%LD W60.11  ; IHM Botão Liga/Desliga todos servos
AND W3.00  ; Flag Inicialização Completa
ORLD
ANDNOT NCx8x_00_Axis3Status_ServoONFlag  ; ServoONFlag
OUT NCx8x_00_Axis3ManualOperation_ServoLockBit  ; ServoLockBit
; rung 1: Unlock Servo
LD AUX_MANUAL  ; auxiliar maquina em trabalho manual
@AND AUX_MANUAL_SERVO_SEL_UNLOCK  ; Auxiliar para UNLOCK Servo SEL
@LD W60.11  ; IHM Botão Liga/Desliga todos servos
AND W3.00  ; Flag Inicialização Completa
ORLD
AND NCx8x_00_Axis3Status_ServoONFlag  ; ServoONFlag
OUT NCx8x_00_Axis3ManualOperation_ServoUnlockBit  ; ServoUnlockBit
; rung 2: Jog Horário
LD AUX_MANUAL  ; auxiliar maquina em trabalho manual
AND W20.07  ; Auxiliar JOG SEL Horario
AND NCx8x_00_Axis3Status_ServoONFlag  ; ServoONFlag
OUT NCx8x_00_Axis3ManualOperation_ForwardJogging_InchingBit  ; ForwardJogging_InchingBit
; rung 3: Jog Anti-Horário
LD AUX_MANUAL  ; auxiliar maquina em trabalho manual
AND W20.08  ; Auxiliar JOG SEL Anti horario
AND NCx8x_00_Axis3Status_ServoONFlag  ; ServoONFlag
OUT NCx8x_00_Axis3ManualOperation_ReverseJogging_InchingBit  ; ReverseJogging_InchingBit
; rung 4
LD P_On
CALL Vel_Selagem : Calc_Vel (Vel_Maq := D410, K_Constante := D403, Vel_Servo => NCx8x_00_Axis3DirectOperation_CommandSpeed)  ; IHM Velocidade Maquina M/min, IHM Constante selagem, CommandSpeed

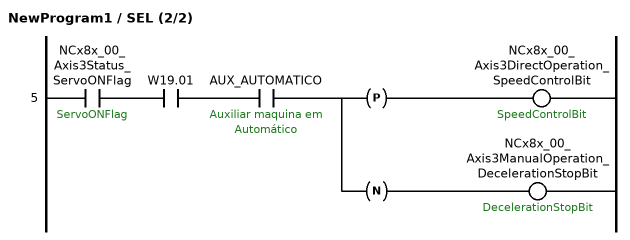
; rung 5
LD NCx8x_00_Axis3Status_ServoONFlag  ; ServoONFlag
AND W19.01
AND AUX_AUTOMATICO  ; Auxiliar maquina em Automático
OUT TR0
UP(521)
OUT NCx8x_00_Axis3DirectOperation_SpeedControlBit  ; SpeedControlBit
LD TR0
DOWN(522)
OUT NCx8x_00_Axis3ManualOperation_DecelerationStopBit  ; DecelerationStopBit

### Section Saídas

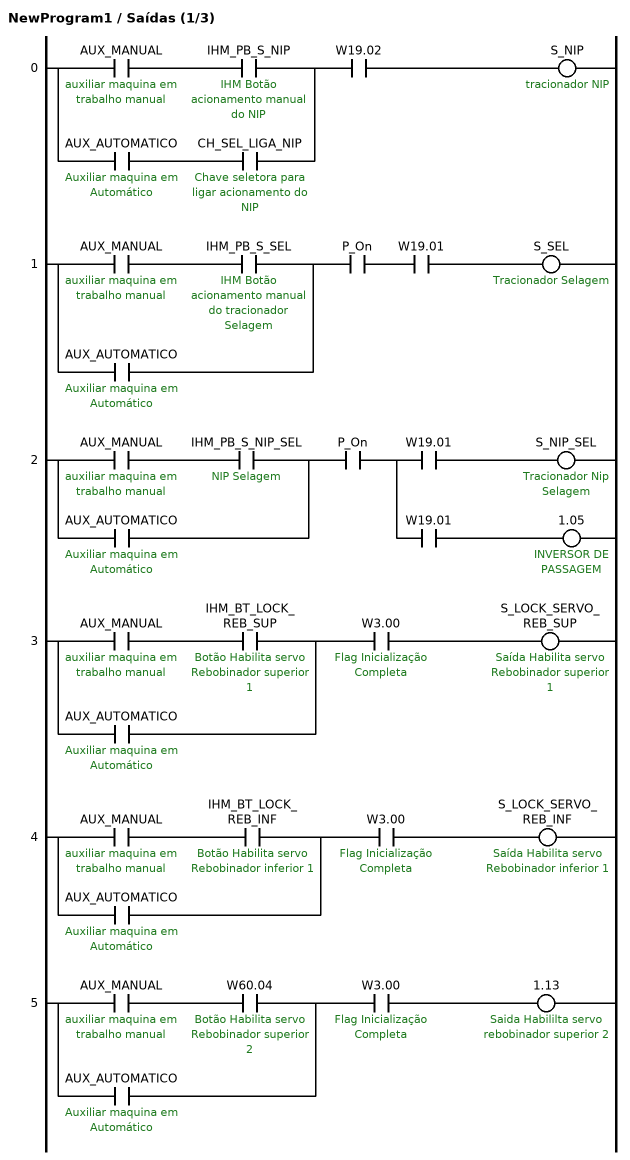
; rung 0
LD AUX_MANUAL  ; auxiliar maquina em trabalho manual
AND IHM_PB_S_NIP  ; IHM Botão acionamento manual do NIP
LD AUX_AUTOMATICO  ; Auxiliar maquina em Automático
AND CH_SEL_LIGA_NIP  ; Chave seletora para ligar acionamento do NIP
ORLD
AND W19.02
OUT S_NIP  ; tracionador NIP
; rung 1
LD AUX_MANUAL  ; auxiliar maquina em trabalho manual
AND IHM_PB_S_SEL  ; IHM Botão acionamento manual do tracionador Selagem
OR AUX_AUTOMATICO  ; Auxiliar maquina em Automático
AND P_On
AND W19.01
OUT S_SEL  ; Tracionador Selagem
; rung 2
LD AUX_MANUAL  ; auxiliar maquina em trabalho manual
AND IHM_PB_S_NIP_SEL  ; NIP Selagem
OR AUX_AUTOMATICO  ; Auxiliar maquina em Automático
AND P_On
OUT TR0
AND W19.01
OUT S_NIP_SEL  ; Tracionador Nip Selagem
LD TR0
AND W19.01
OUT 1.05  ; INVERSOR DE PASSAGEM
; rung 3
LD AUX_MANUAL  ; auxiliar maquina em trabalho manual
AND IHM_BT_LOCK_REB_SUP  ; Botão Habilita servo Rebobinador superior 1
OR AUX_AUTOMATICO  ; Auxiliar maquina em Automático
AND W3.00  ; Flag Inicialização Completa
OUT S_LOCK_SERVO_REB_SUP  ; Saída Habilita servo Rebobinador superior 1
; rung 4
LD AUX_MANUAL  ; auxiliar maquina em trabalho manual
AND IHM_BT_LOCK_REB_INF  ; Botão Habilita servo Rebobinador inferior 1
OR AUX_AUTOMATICO  ; Auxiliar maquina em Automático
AND W3.00  ; Flag Inicialização Completa
OUT S_LOCK_SERVO_REB_INF  ; Saída Habilita servo Rebobinador inferior 1
; rung 5
LD AUX_MANUAL  ; auxiliar maquina em trabalho manual
AND W60.04  ; Botão Habilita servo Rebobinador superior 2
OR AUX_AUTOMATICO  ; Auxiliar maquina em Automático
AND W3.00  ; Flag Inicialização Completa
OUT 1.13  ; Saida Habililta servo rebobinador superior 2

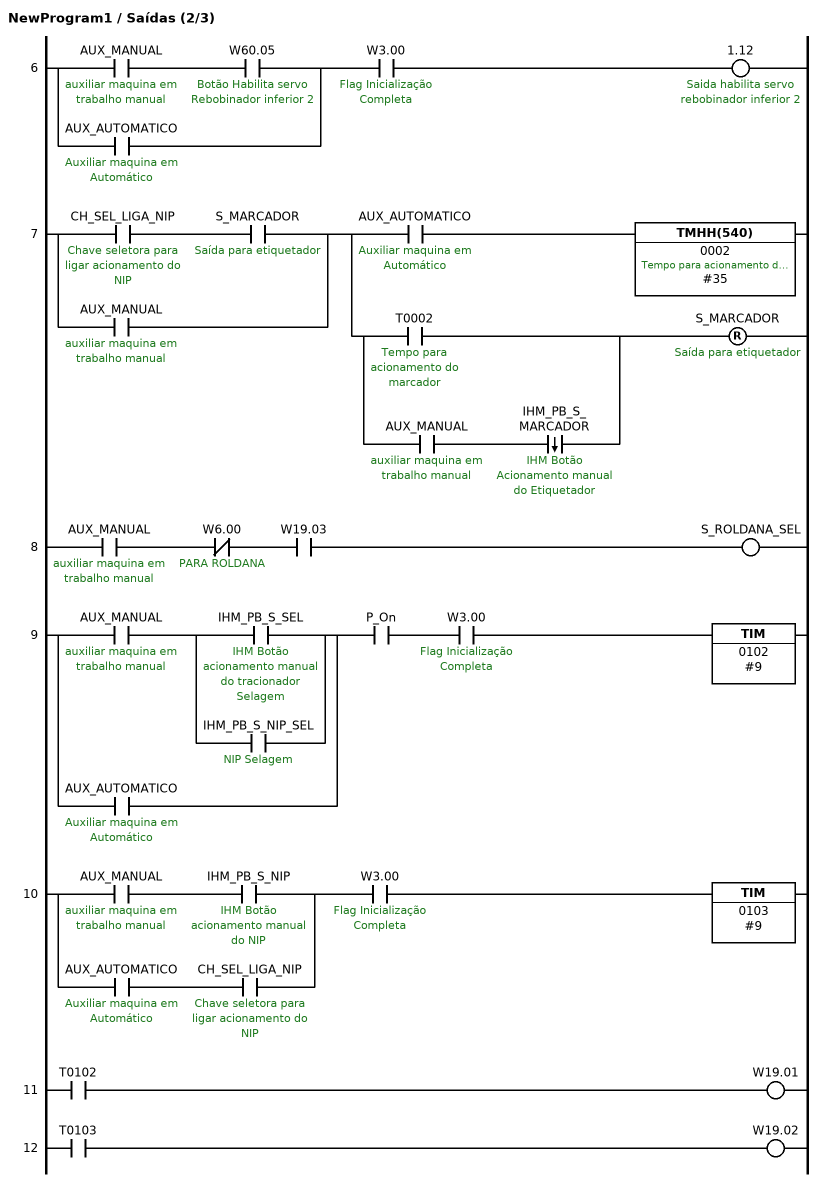
; rung 6
LD AUX_MANUAL  ; auxiliar maquina em trabalho manual
AND W60.05  ; Botão Habilita servo Rebobinador inferior 2
OR AUX_AUTOMATICO  ; Auxiliar maquina em Automático
AND W3.00  ; Flag Inicialização Completa
OUT 1.12  ; Saida habilita servo rebobinador inferior 2
; rung 7
LD CH_SEL_LIGA_NIP  ; Chave seletora para ligar acionamento do NIP
AND S_MARCADOR  ; Saída para etiquetador
OR AUX_MANUAL  ; auxiliar maquina em trabalho manual
OUT TR0
AND AUX_AUTOMATICO  ; Auxiliar maquina em Automático
TMHH(540) 0002 #35  ; Tempo para acionamento do marcador
LD TR0
LD T0002  ; Tempo para acionamento do marcador
LD AUX_MANUAL  ; auxiliar maquina em trabalho manual
%AND IHM_PB_S_MARCADOR  ; IHM Botão Acionamento manual do Etiquetador
ORLD
ANDLD
RSET S_MARCADOR  ; Saída para etiquetador
; rung 8
LD AUX_MANUAL  ; auxiliar maquina em trabalho manual
ANDNOT W6.00  ; PARA ROLDANA
AND W19.03
OUT S_ROLDANA_SEL
; rung 9
LD AUX_MANUAL  ; auxiliar maquina em trabalho manual
LD IHM_PB_S_SEL  ; IHM Botão acionamento manual do tracionador Selagem
OR IHM_PB_S_NIP_SEL  ; NIP Selagem
ANDLD
OR AUX_AUTOMATICO  ; Auxiliar maquina em Automático
AND P_On
AND W3.00  ; Flag Inicialização Completa
TIM 0102 #9
; rung 10
LD AUX_MANUAL  ; auxiliar maquina em trabalho manual
AND IHM_PB_S_NIP  ; IHM Botão acionamento manual do NIP
LD AUX_AUTOMATICO  ; Auxiliar maquina em Automático
AND CH_SEL_LIGA_NIP  ; Chave seletora para ligar acionamento do NIP
ORLD
AND W3.00  ; Flag Inicialização Completa
TIM 0103 #9
; rung 11
LD T0102
OUT W19.01
; rung 12
LD T0103
OUT W19.02

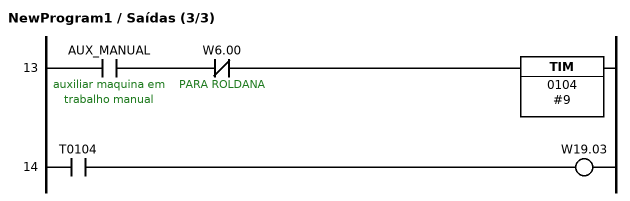
; rung 13
LD AUX_MANUAL  ; auxiliar maquina em trabalho manual
ANDNOT W6.00  ; PARA ROLDANA
TIM 0104 #9
; rung 14
LD T0104
OUT W19.03

### Section Manual

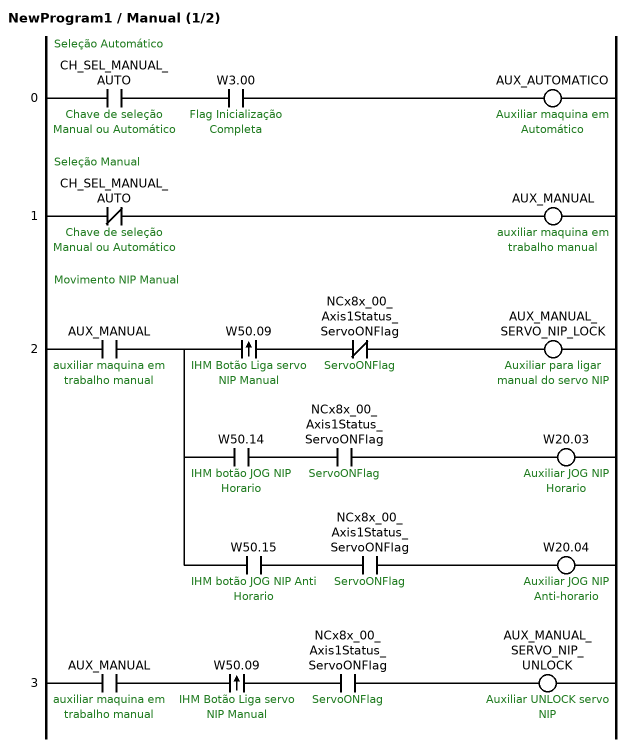
; rung 0: Seleção Automático
LD CH_SEL_MANUAL_AUTO  ; Chave de seleção Manual ou Automático
AND W3.00  ; Flag Inicialização Completa
OUT AUX_AUTOMATICO  ; Auxiliar maquina em Automático
; rung 1: Seleção Manual
LDNOT CH_SEL_MANUAL_AUTO  ; Chave de seleção Manual ou Automático
OUT AUX_MANUAL  ; auxiliar maquina em trabalho manual
; rung 2: Movimento NIP Manual
LD AUX_MANUAL  ; auxiliar maquina em trabalho manual
OUT TR0
@AND W50.09  ; IHM Botão Liga servo NIP Manual
ANDNOT NCx8x_00_Axis1Status_ServoONFlag  ; ServoONFlag
OUT AUX_MANUAL_SERVO_NIP_LOCK  ; Auxiliar para ligar manual do servo NIP
LD TR0
AND W50.14  ; IHM botão JOG NIP Horario
AND NCx8x_00_Axis1Status_ServoONFlag  ; ServoONFlag
OUT W20.03  ; Auxiliar JOG NIP Horario
LD TR0
AND W50.15  ; IHM botão JOG NIP Anti Horario
AND NCx8x_00_Axis1Status_ServoONFlag  ; ServoONFlag
OUT W20.04  ; Auxiliar JOG NIP Anti-horario
; rung 3
LD AUX_MANUAL  ; auxiliar maquina em trabalho manual
@AND W50.09  ; IHM Botão Liga servo NIP Manual
AND NCx8x_00_Axis1Status_ServoONFlag  ; ServoONFlag
OUT AUX_MANUAL_SERVO_NIP_UNLOCK  ; Auxiliar UNLOCK servo NIP

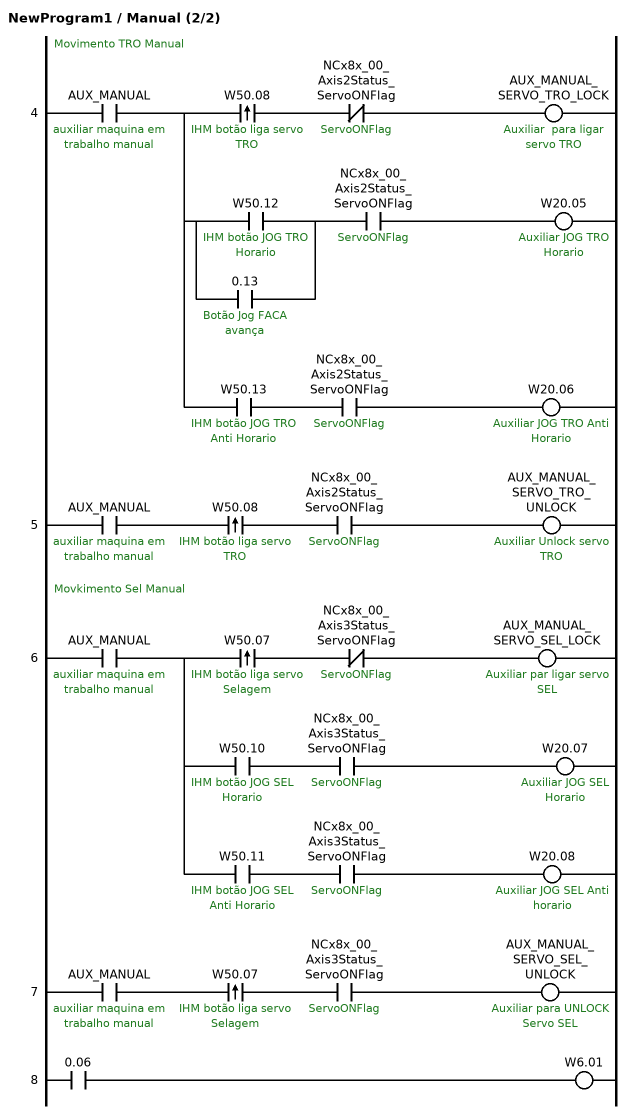
; rung 4: Movimento TRO Manual
LD AUX_MANUAL  ; auxiliar maquina em trabalho manual
OUT TR0
@AND W50.08  ; IHM botão liga servo TRO
ANDNOT NCx8x_00_Axis2Status_ServoONFlag  ; ServoONFlag
OUT AUX_MANUAL_SERVO_TRO_LOCK  ; Auxiliar  para ligar servo TRO
LD TR0
LD W50.12  ; IHM botão JOG TRO Horario
OR 0.13  ; Botão Jog FACA avança
ANDLD
AND NCx8x_00_Axis2Status_ServoONFlag  ; ServoONFlag
OUT W20.05  ; Auxiliar JOG TRO Horario
LD TR0
AND W50.13  ; IHM botão JOG TRO Anti Horario
AND NCx8x_00_Axis2Status_ServoONFlag  ; ServoONFlag
OUT W20.06  ; Auxiliar JOG TRO Anti Horario
; rung 5
LD AUX_MANUAL  ; auxiliar maquina em trabalho manual
@AND W50.08  ; IHM botão liga servo TRO
AND NCx8x_00_Axis2Status_ServoONFlag  ; ServoONFlag
OUT AUX_MANUAL_SERVO_TRO_UNLOCK  ; Auxiliar Unlock servo TRO
; rung 6: Movkimento Sel Manual
LD AUX_MANUAL  ; auxiliar maquina em trabalho manual
OUT TR0
@AND W50.07  ; IHM botão liga servo Selagem
ANDNOT NCx8x_00_Axis3Status_ServoONFlag  ; ServoONFlag
OUT AUX_MANUAL_SERVO_SEL_LOCK  ; Auxiliar par ligar servo SEL
LD TR0
AND W50.10  ; IHM botão JOG SEL Horario
AND NCx8x_00_Axis3Status_ServoONFlag  ; ServoONFlag
OUT W20.07  ; Auxiliar JOG SEL Horario
LD TR0
AND W50.11  ; IHM botão JOG SEL Anti Horario
AND NCx8x_00_Axis3Status_ServoONFlag  ; ServoONFlag
OUT W20.08  ; Auxiliar JOG SEL Anti horario
; rung 7
LD AUX_MANUAL  ; auxiliar maquina em trabalho manual
@AND W50.07  ; IHM botão liga servo Selagem
AND NCx8x_00_Axis3Status_ServoONFlag  ; ServoONFlag
OUT AUX_MANUAL_SERVO_SEL_UNLOCK  ; Auxiliar para UNLOCK Servo SEL
; rung 8
LD 0.06
OUT W6.01

### Section Rebobinador_Sup

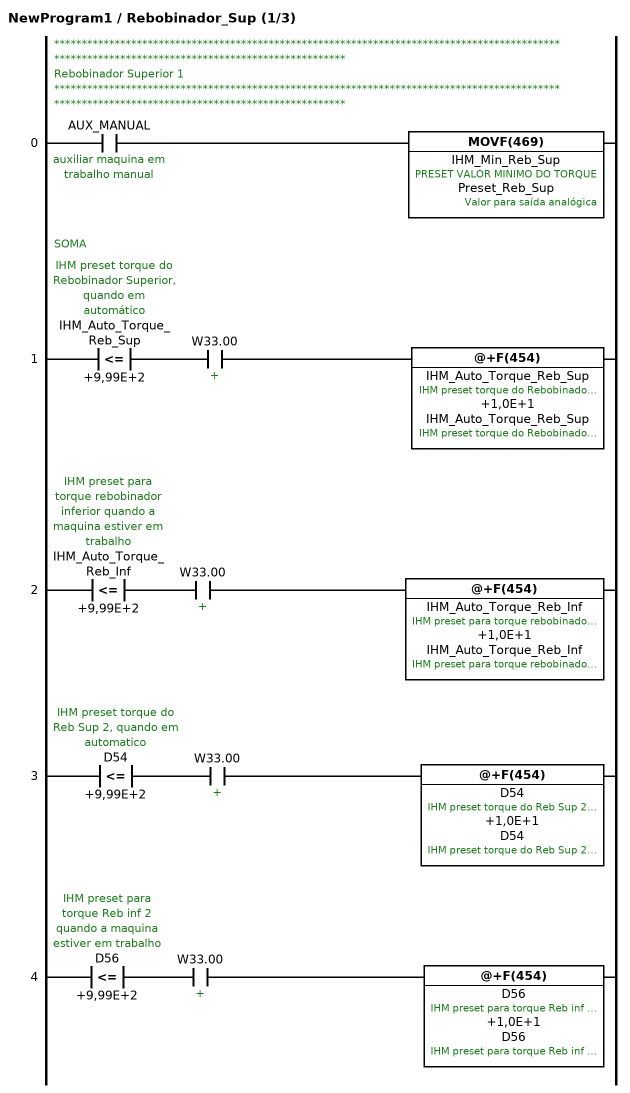
; rung 0: ************************************************************************************************************************************************* / Rebobinador Superior 1 / *************************************************************************************************************************************************
LD AUX_MANUAL  ; auxiliar maquina em trabalho manual
MOVF(469) IHM_Min_Reb_Sup Preset_Reb_Sup  ; PRESET VALOR MINIMO DO TORQUE, Valor para saída analógica
; rung 1: SOMA
LD<=F(332) IHM_Auto_Torque_Reb_Sup +9,99E+2  ; IHM preset torque do Rebobinador Superior, quando em automático
AND W33.00  ; +
@+F(454) IHM_Auto_Torque_Reb_Sup +1,0E+1 IHM_Auto_Torque_Reb_Sup  ; IHM preset torque do Rebobinador Superior, quando em automático
; rung 2
LD<=F(332) IHM_Auto_Torque_Reb_Inf +9,99E+2  ; IHM preset para torque rebobinador inferior quando a maquina estiver em trabalho
AND W33.00  ; +
@+F(454) IHM_Auto_Torque_Reb_Inf +1,0E+1 IHM_Auto_Torque_Reb_Inf  ; IHM preset para torque rebobinador inferior quando a maquina estiver em trabalho
; rung 3
LD<=F(332) D54 +9,99E+2  ; IHM preset torque do Reb Sup 2, quando em automatico
AND W33.00  ; +
@+F(454) D54 +1,0E+1 D54  ; IHM preset torque do Reb Sup 2, quando em automatico
; rung 4
LD<=F(332) D56 +9,99E+2  ; IHM preset para torque Reb inf 2 quando a maquina estiver em trabalho
AND W33.00  ; +
@+F(454) D56 +1,0E+1 D56  ; IHM preset para torque Reb inf 2 quando a maquina estiver em trabalho

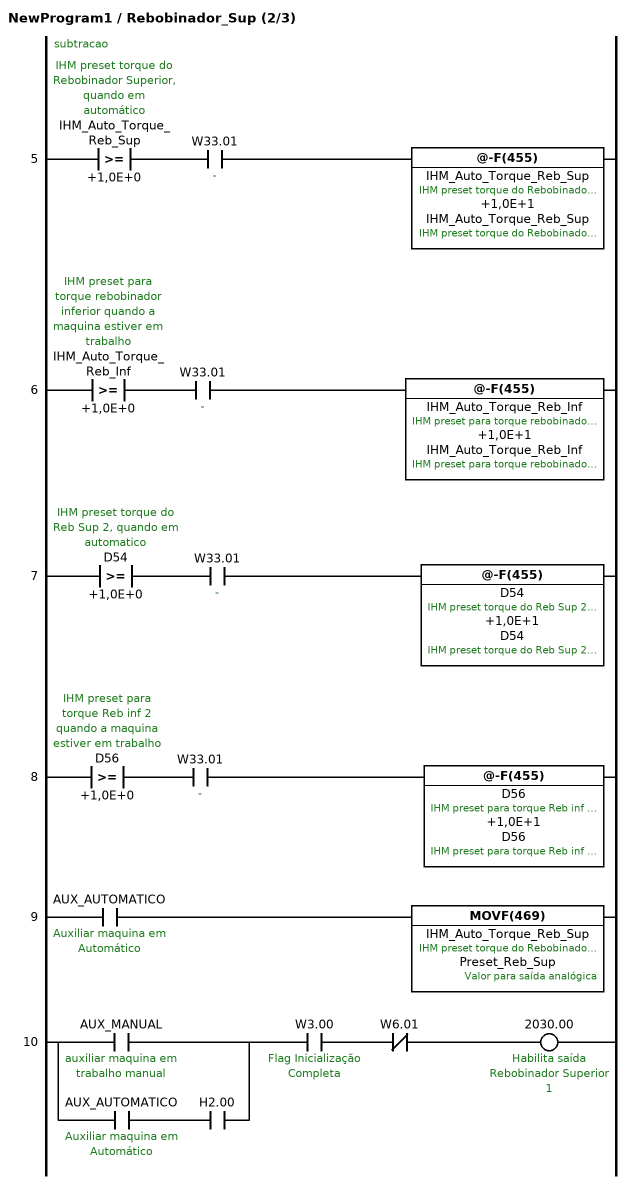
; rung 5: subtracao
LD>=F(334) IHM_Auto_Torque_Reb_Sup +1,0E+0  ; IHM preset torque do Rebobinador Superior, quando em automático
AND W33.01  ; -
@-F(455) IHM_Auto_Torque_Reb_Sup +1,0E+1 IHM_Auto_Torque_Reb_Sup  ; IHM preset torque do Rebobinador Superior, quando em automático
; rung 6
LD>=F(334) IHM_Auto_Torque_Reb_Inf +1,0E+0  ; IHM preset para torque rebobinador inferior quando a maquina estiver em trabalho
AND W33.01  ; -
@-F(455) IHM_Auto_Torque_Reb_Inf +1,0E+1 IHM_Auto_Torque_Reb_Inf  ; IHM preset para torque rebobinador inferior quando a maquina estiver em trabalho
; rung 7
LD>=F(334) D54 +1,0E+0  ; IHM preset torque do Reb Sup 2, quando em automatico
AND W33.01  ; -
@-F(455) D54 +1,0E+1 D54  ; IHM preset torque do Reb Sup 2, quando em automatico
; rung 8
LD>=F(334) D56 +1,0E+0  ; IHM preset para torque Reb inf 2 quando a maquina estiver em trabalho
AND W33.01  ; -
@-F(455) D56 +1,0E+1 D56  ; IHM preset para torque Reb inf 2 quando a maquina estiver em trabalho
; rung 9
LD AUX_AUTOMATICO  ; Auxiliar maquina em Automático
MOVF(469) IHM_Auto_Torque_Reb_Sup Preset_Reb_Sup  ; IHM preset torque do Rebobinador Superior, quando em automático, Valor para saída analógica
; rung 10
LD AUX_MANUAL  ; auxiliar maquina em trabalho manual
LD AUX_AUTOMATICO  ; Auxiliar maquina em Automático
AND H2.00
ORLD
AND W3.00  ; Flag Inicialização Completa
ANDNOT W6.01
OUT 2030.00  ; Habilita saída Rebobinador Superior 1

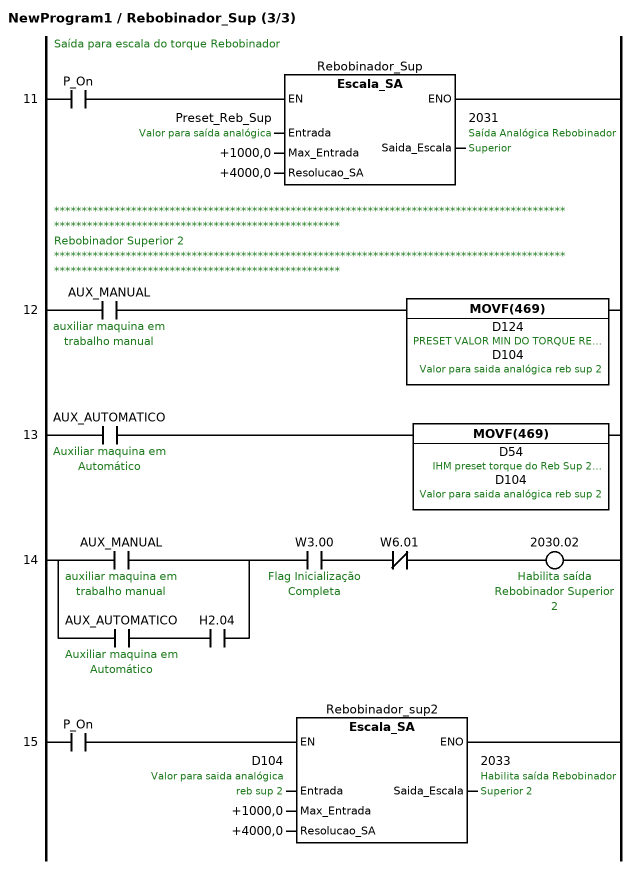
; rung 11: Saída para escala do torque Rebobinador
LD P_On
CALL Rebobinador_Sup : Escala_SA (Entrada := Preset_Reb_Sup, Max_Entrada := +1000,0, Resolucao_SA := +4000,0, Saida_Escala => 2031)  ; Valor para saída analógica, Saída Analógica Rebobinador Superior
; rung 12: ************************************************************************************************************************************************* / Rebobinador Superior 2 / *************************************************************************************************************************************************
LD AUX_MANUAL  ; auxiliar maquina em trabalho manual
MOVF(469) D124 D104  ; PRESET VALOR MIN DO TORQUE REB SUP 2, Valor para saida analógica reb sup 2
; rung 13
LD AUX_AUTOMATICO  ; Auxiliar maquina em Automático
MOVF(469) D54 D104  ; IHM preset torque do Reb Sup 2, quando em automatico, Valor para saida analógica reb sup 2
; rung 14
LD AUX_MANUAL  ; auxiliar maquina em trabalho manual
LD AUX_AUTOMATICO  ; Auxiliar maquina em Automático
AND H2.04
ORLD
AND W3.00  ; Flag Inicialização Completa
ANDNOT W6.01
OUT 2030.02  ; Habilita saída Rebobinador Superior 2
; rung 15
LD P_On
CALL Rebobinador_sup2 : Escala_SA (Entrada := D104, Max_Entrada := +1000,0, Resolucao_SA := +4000,0, Saida_Escala => 2033)  ; Valor para saida analógica reb sup 2, Habilita saída Rebobinador Superior 2

### Section Rebobinador_Inf

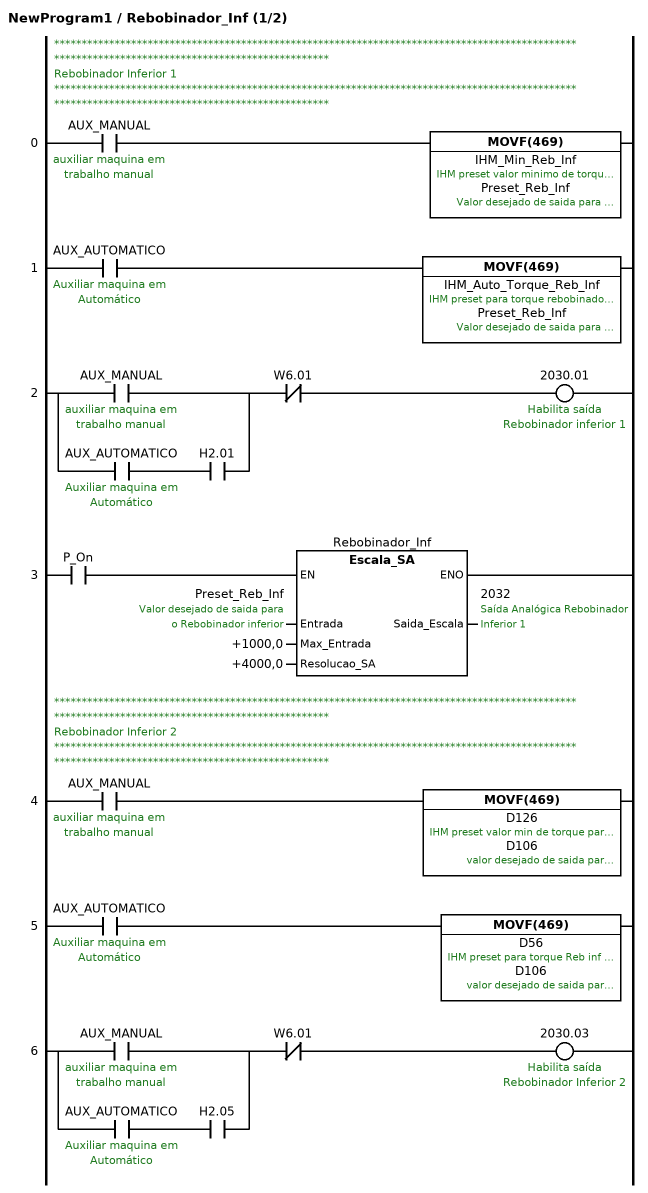
; rung 0: ************************************************************************************************************************************************* / Rebobinador Inferior 1 / *************************************************************************************************************************************************
LD AUX_MANUAL  ; auxiliar maquina em trabalho manual
MOVF(469) IHM_Min_Reb_Inf Preset_Reb_Inf  ; IHM preset valor minimo de torque para trabalho, Valor desejado de saida para o Rebobinador inferior
; rung 1
LD AUX_AUTOMATICO  ; Auxiliar maquina em Automático
MOVF(469) IHM_Auto_Torque_Reb_Inf Preset_Reb_Inf  ; IHM preset para torque rebobinador inferior quando a maquina estiver em trabalho, Valor desejado de saida para o Rebobinador inferior
; rung 2
LD AUX_MANUAL  ; auxiliar maquina em trabalho manual
LD AUX_AUTOMATICO  ; Auxiliar maquina em Automático
AND H2.01
ORLD
ANDNOT W6.01
OUT 2030.01  ; Habilita saída Rebobinador inferior 1
; rung 3
LD P_On
CALL Rebobinador_Inf : Escala_SA (Entrada := Preset_Reb_Inf, Max_Entrada := +1000,0, Resolucao_SA := +4000,0, Saida_Escala => 2032)  ; Valor desejado de saida para o Rebobinador inferior, Saída Analógica Rebobinador  Inferior 1
; rung 4: ************************************************************************************************************************************************* / Rebobinador Inferior 2 / *************************************************************************************************************************************************
LD AUX_MANUAL  ; auxiliar maquina em trabalho manual
MOVF(469) D126 D106  ; IHM preset valor min de torque para trabalho inferior2, valor desejado de saida para rebobinador inferior 2
; rung 5
LD AUX_AUTOMATICO  ; Auxiliar maquina em Automático
MOVF(469) D56 D106  ; IHM preset para torque Reb inf 2 quando a maquina estiver em trabalho, valor desejado de saida para rebobinador inferior 2
; rung 6
LD AUX_MANUAL  ; auxiliar maquina em trabalho manual
LD AUX_AUTOMATICO  ; Auxiliar maquina em Automático
AND H2.05
ORLD
ANDNOT W6.01
OUT 2030.03  ; Habilita saída Rebobinador Inferior 2

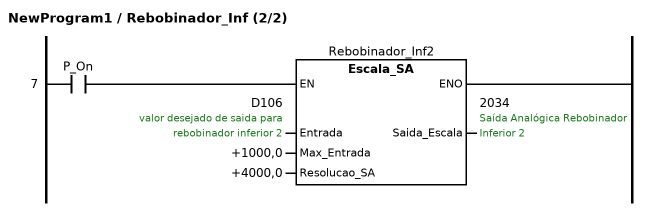
; rung 7
LD P_On
CALL Rebobinador_Inf2 : Escala_SA (Entrada := D106, Max_Entrada := +1000,0, Resolucao_SA := +4000,0, Saida_Escala => 2034)  ; valor desejado de saida para rebobinador inferior 2, Saída Analógica Rebobinador  Inferior 2

### Section Desbobinador_Sup

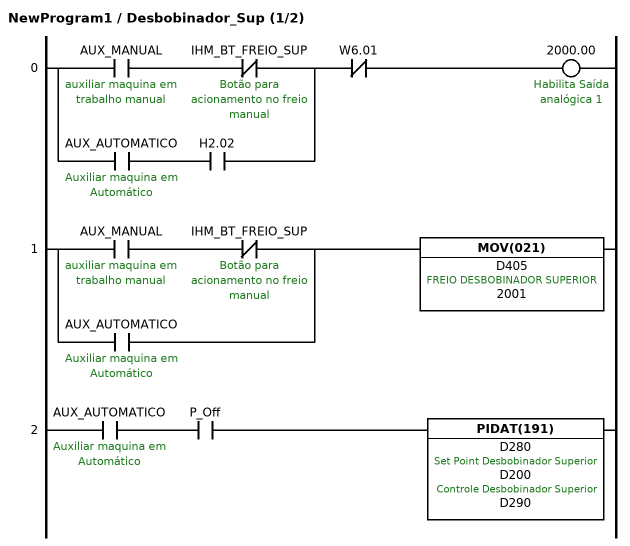
; rung 0
LD AUX_MANUAL  ; auxiliar maquina em trabalho manual
ANDNOT IHM_BT_FREIO_SUP  ; Botão para acionamento no freio manual
LD AUX_AUTOMATICO  ; Auxiliar maquina em Automático
AND H2.02
ORLD
ANDNOT W6.01
OUT 2000.00  ; Habilita Saída analógica 1
; rung 1
LD AUX_MANUAL  ; auxiliar maquina em trabalho manual
ANDNOT IHM_BT_FREIO_SUP  ; Botão para acionamento no freio manual
OR AUX_AUTOMATICO  ; Auxiliar maquina em Automático
MOV(021) D405 2001  ; FREIO DESBOBINADOR SUPERIOR
; rung 2
LD AUX_AUTOMATICO  ; Auxiliar maquina em Automático
AND P_Off
PIDAT(191) D280 D200 D290  ; Set Point Desbobinador Superior, Controle Desbobinador Superior

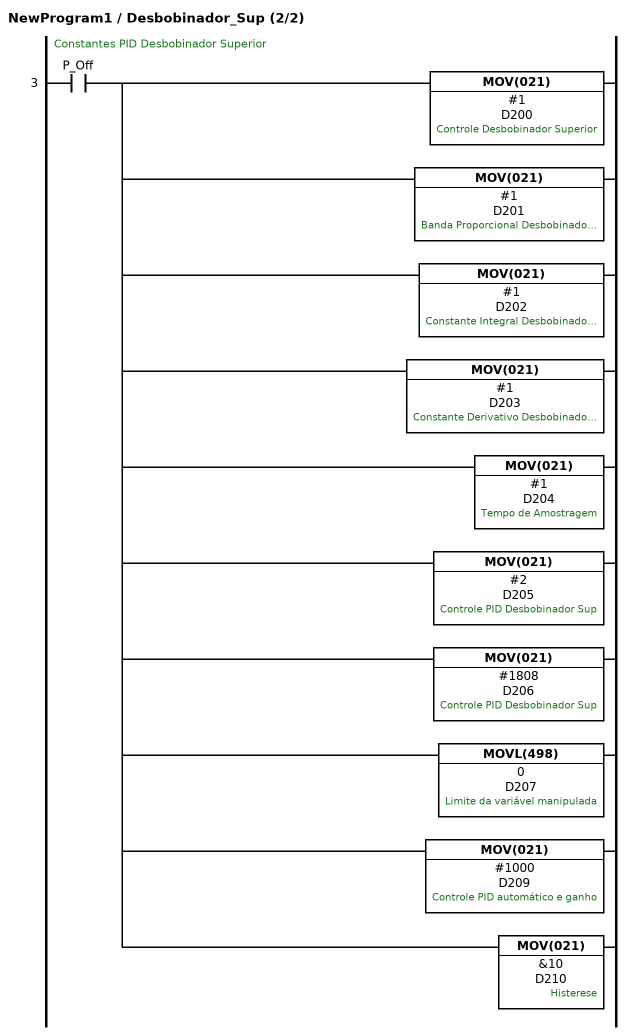
; rung 3: Constantes PID Desbobinador Superior
LD P_Off
MOV(021) #1 D200  ; Controle Desbobinador Superior
MOV(021) #1 D201  ; Banda Proporcional Desbobinador superior
MOV(021) #1 D202  ; Constante Integral Desbobinador Superior
MOV(021) #1 D203  ; Constante Derivativo Desbobinador Superior
MOV(021) #1 D204  ; Tempo de Amostragem
MOV(021) #2 D205  ; Controle PID Desbobinador Sup  // Controle PID / Bit 0 - 0=Reverse, 1=Forward / Bit 1 - 0=Alteração das constantes na execução da instrução, 1=Alteração das constantes no tempo de amostragem / Bit 2 - 0 / Bit 3 - 0=Manipulação da Variávem em 0% quando PV=SV, 1=Manipulação da variável em 50% quando PV=SV / Bit 4 até 15 - Coeficiente do filtro
MOV(021) #1808 D206  ; Controle PID Desbobinador Sup  // Controle PID / Bit 0 até 3 - qntidade bits na saída / Bit 4 até 7 - unidade do  periodo para amostragem / Bit 8 até 11 - Range da entrada / Bit 12 - 0= desabilita limite para variável manipulada, 1=Habilita limite para variável manipulada / Bit 13 até 14 - Deteermina o valor inicial para o valor integral qndo inicio do PID
MOVL(498) 0 D207  ; Limite da variável manipulada
MOV(021) #1000 D209  ; Controle PID automático e ganho  // Bit 0 até 11 - Controle do ganho / Bit 15 - 0=Desliga Auto Tune, 1=Habilita Auto Tune
MOV(021) &10 D210  ; Histerese

### Section Desbobinador_Inf

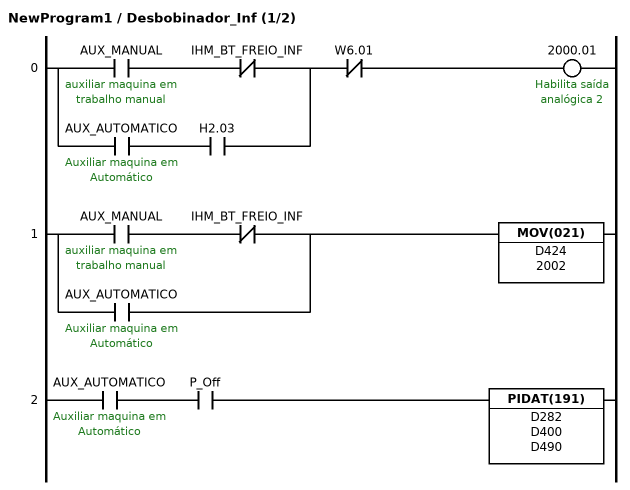
; rung 0
LD AUX_MANUAL  ; auxiliar maquina em trabalho manual
ANDNOT IHM_BT_FREIO_INF
LD AUX_AUTOMATICO  ; Auxiliar maquina em Automático
AND H2.03
ORLD
ANDNOT W6.01
OUT 2000.01  ; Habilita saída analógica 2
; rung 1
LD AUX_MANUAL  ; auxiliar maquina em trabalho manual
ANDNOT IHM_BT_FREIO_INF
OR AUX_AUTOMATICO  ; Auxiliar maquina em Automático
MOV(021) D424 2002
; rung 2
LD AUX_AUTOMATICO  ; Auxiliar maquina em Automático
AND P_Off
PIDAT(191) D282 D400 D490

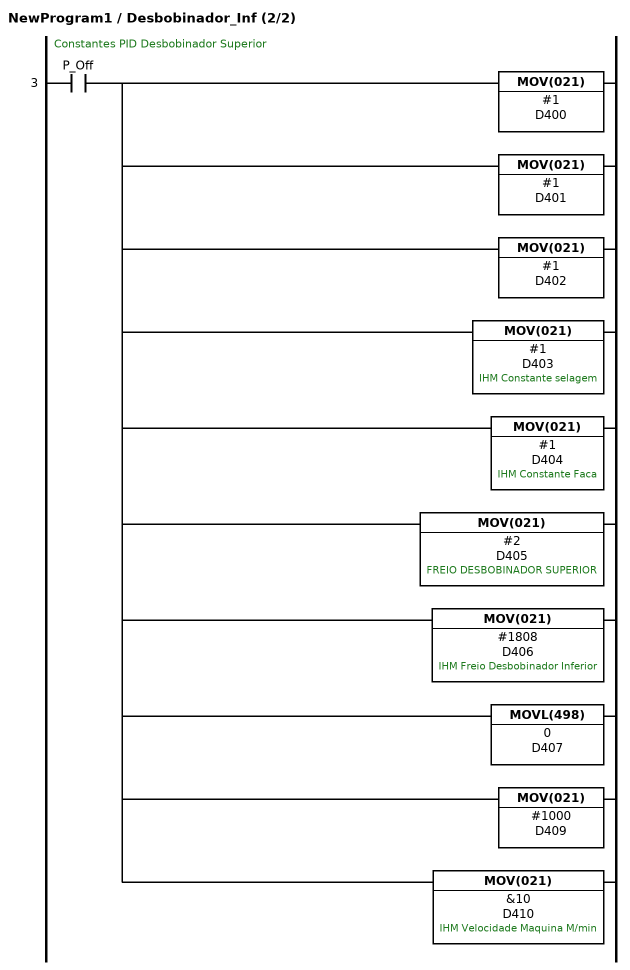
; rung 3: Constantes PID Desbobinador Superior
LD P_Off
MOV(021) #1 D400
MOV(021) #1 D401
MOV(021) #1 D402
MOV(021) #1 D403  ; IHM Constante selagem
MOV(021) #1 D404  ; IHM Constante Faca
MOV(021) #2 D405  ; FREIO DESBOBINADOR SUPERIOR  // Controle PID / Bit 0 - 0=Reverse, 1=Forward / Bit 1 - 0=Alteração das constantes na execução da instrução, 1=Alteração das constantes no tempo de amostragem / Bit 2 - 0 / Bit 3 - 0=Manipulação da Variávem em 0% quando PV=SV, 1=Manipulação da variável em 50% quando PV=SV / Bit 4 até 15 - Coeficiente do filtro
MOV(021) #1808 D406  ; IHM Freio Desbobinador Inferior  // Controle PID / Bit 0 até 3 - qntidade bits na saída / Bit 4 até 7 - unidade do  periodo para amostragem / Bit 8 até 11 - Range da entrada / Bit 12 - 0= desabilita limite para variável manipulada, 1=Habilita limite para variável manipulada / Bit 13 até 14 - Deteermina o valor inicial para o valor integral qndo inicio do PID
MOVL(498) 0 D407
MOV(021) #1000 D409  // Bit 0 até 11 - Controle do ganho / Bit 15 - 0=Desliga Auto Tune, 1=Habilita Auto Tune
MOV(021) &10 D410  ; IHM Velocidade Maquina M/min

### Section Inicialização

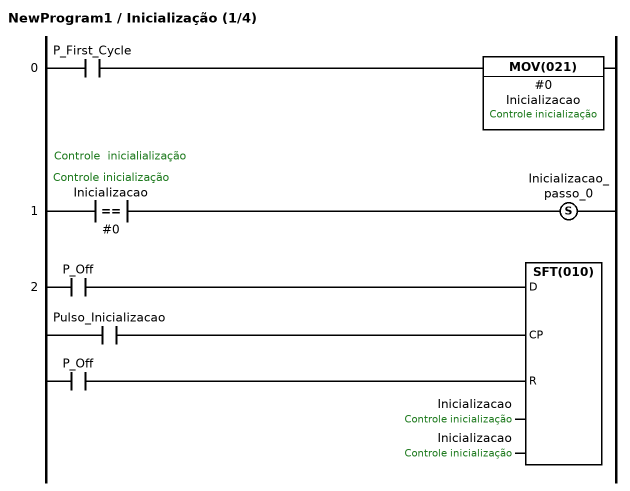
; rung 0
LD P_First_Cycle
MOV(021) #0 Inicializacao  ; Controle inicialização
; rung 1: Controle  inicialialização
LD=(300) Inicializacao #0  ; Controle inicialização
SET Inicializacao_passo_0
; rung 2
LD P_Off
LD Pulso_Inicializacao
LD P_Off
SFT(010) Inicializacao Inicializacao  ; Controle inicialização

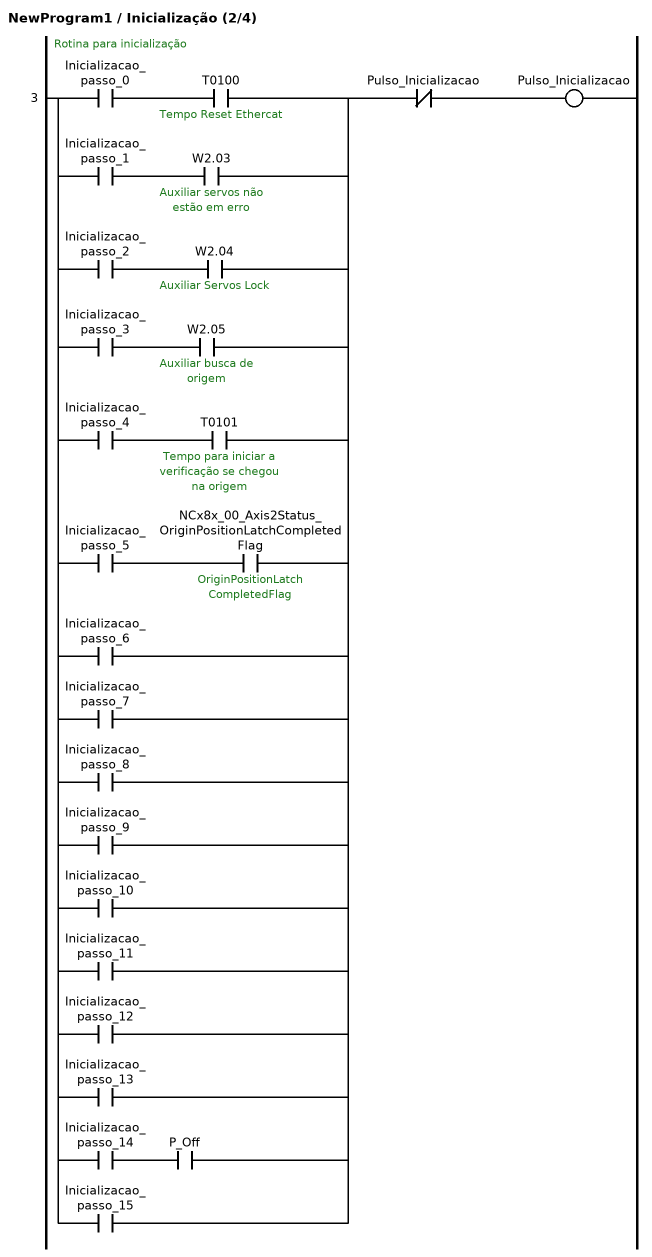
; rung 3: Rotina para inicialização
LD Inicializacao_passo_0
AND T0100  ; Tempo Reset Ethercat
LD Inicializacao_passo_1
AND W2.03  ; Auxiliar servos não estão em erro
ORLD
LD Inicializacao_passo_2
AND W2.04  ; Auxiliar Servos Lock
ORLD
LD Inicializacao_passo_3
AND W2.05  ; Auxiliar busca de origem
ORLD
LD Inicializacao_passo_4
AND T0101  ; Tempo para iniciar a verificação se chegou na origem
ORLD
LD Inicializacao_passo_5
AND NCx8x_00_Axis2Status_OriginPositionLatchCompletedFlag  ; OriginPositionLatchCompletedFlag
ORLD
OR Inicializacao_passo_6
OR Inicializacao_passo_7
OR Inicializacao_passo_8
OR Inicializacao_passo_9
OR Inicializacao_passo_10
OR Inicializacao_passo_11
OR Inicializacao_passo_12
OR Inicializacao_passo_13
LD Inicializacao_passo_14
AND P_Off
ORLD
OR Inicializacao_passo_15
ANDNOT Pulso_Inicializacao
OUT Pulso_Inicializacao

